LIN {X 0,Y 524.198,Z 429.088,A -85,B 0,C 180,E1 -4760.353,E2 -4760.353} C_VEL
LIN {X 0,Y 524.005,Z 439.005,A -85,B 0,C 180,E1 -4761.03,E2 -4761.03} C_VEL
LIN {X 0,Y 523.832,Z 446.958,A -85,B 0,C 180,E1 -4761.708,E2 -4761.708} C_VEL
LIN {X 0,Y 523.699,Z 454.397,A -85,B 0,C 180,E1 -4762.482,E2 -4762.482} C_VEL
LIN {X 0,Y 523.622,Z 461.025,A -85,B 0,C 180,E1 -4763.324,E2 -4763.324} C_VEL
LIN {X 0,Y 523.51,Z 467.877,A -85,B 0,C 180,E1 -4764.415,E2 -4764.415} C_VEL
LIN {X 0,Y 523.401,Z 472.538,A -85,B 0,C 180,E1 -4765.379,E2 -4765.379} C_VEL
LIN {X 0,Y 523.454,Z 475.573,A -85,B 0,C 180,E1 -4766.151,E2 -4766.151} C_VEL
LIN {X 0,Y 523.38,Z 477.92,A -85,B 0,C 180,E1 -4766.921,E2 -4766.921} C_VEL
LIN {X 0,Y 523.336,Z 479.685,A -85,B 0,C 180,E1 -4767.691,E2 -4767.691} C_VEL
LIN {X 0,Y 523.273,Z 480.952,A -85,B 0,C 180,E1 -4768.461,E2 -4768.461} C_VEL
LIN {X 0,Y 523.261,Z 481.745,A -85,B 0,C 180,E1 -4769.231,E2 -4769.231} C_VEL
LIN {X 0,Y 523.264,Z 482.047,A -85,B 0,C 180,E1 -4770,E2 -4770} C_VEL
LIN {X 0,Y 523.26,Z 481.751,A -85,B 0,C 180,E1 -4770.77,E2 -4770.77} C_VEL
LIN {X 0,Y 523.273,Z 480.966,A -85,B 0,C 180,E1 -4771.539,E2 -4771.539} C_VEL
LIN {X 0,Y 523.336,Z 479.706,A -85,B 0,C 180,E1 -4772.309,E2 -4772.309} C_VEL
LIN {X 0,Y 523.407,Z 476.783,A -85,B 0,C 180,E1 -4773.464,E2 -4773.464} C_VEL
LIN {X 0,Y 523.451,Z 474.115,A -85,B 0,C 180,E1 -4774.235,E2 -4774.235} C_VEL
LIN {X 0,Y 523.483,Z 468.893,A -85,B 0,C 180,E1 -4775.393,E2 -4775.393} C_VEL
LIN {X 0,Y 523.573,Z 462.971,A -85,B 0,C 180,E1 -4776.408,E2 -4776.408} C_VEL
LIN {X 0,Y 523.699,Z 456.194,A -85,B 0,C 180,E1 -4777.325,E2 -4777.325} C_VEL
LIN {X 0,Y 523.837,Z 448.092,A -85,B 0,C 180,E1 -4778.195,E2 -4778.195} C_VEL
LIN {X 0,Y 524.001,Z 440.358,A -85,B 0,C 180,E1 -4778.873,E2 -4778.873} C_VEL
LIN {X 0,Y 524.123,Z 432.228,A -85,B 0,C 180,E1 -4779.454,E2 -4779.454} C_VEL
LIN {X 0,Y 524.305,Z 423.801,A -85,B 0,C 180,E1 -4779.938,E2 -4779.938} C_VEL
LIN {X 0,Y 524.43,Z 415.18,A -85,B 0,C 180,E1 -4780.326,E2 -4780.326} C_VEL
LIN {X 0,Y 524.599,Z 404.889,A -85,B 0,C 180,E1 -4780.664,E2 -4780.664} C_VEL
LIN {X 0,Y 524.733,Z 390.891,A -85,B 0,C 180,E1 -4780.929,E2 -4780.929} C_VEL
LIN {X 0,Y 524.752,Z 329.083,A -85,B 0,C 180,E1 -4781.779,E2 -4781.779} C_VEL
LIN {X 0,Y 523.843,Z 320.89,A -85,B 0,C 180,E1 -4781.93,E2 -4781.93} C_VEL
LIN {X 0,Y 524.085,Z 303.68,A -85,B 0,C 180,E1 -4784.761,E2 -4784.761} C_VEL
LIN {X 0,Y 524.361,Z 286.918,A -85,B 0,C 180,E1 -4787.532,E2 -4787.532} C_VEL
LIN {X 0,Y 524.693,Z 269.864,A -85,B 0,C 180,E1 -4790.38,E2 -4790.38} C_VEL
LIN {X 0,Y 525.038,Z 257.174,A -85,B 0,C 180,E1 -4792.54,E2 -4792.54} C_VEL
LIN {X 0,Y 523.945,Z 250.036,A -85,B 0,C 180,E1 -4793.834,E2 -4793.834} C_VEL
LIN {X 0,Y 523.94,Z 250.03,A -85,B 0,C 180,E1 -4796.273,E2 -4796.273} C_VEL
LIN {X 0,Y 523.928,Z 250.031,A -85,B 0,C 180,E1 -4798.875,E2 -4798.875} C_VEL
LIN {X 0,Y 523.92,Z 250.04,A -85,B 0,C 180,E1 -4801.544,E2 -4801.544} C_VEL
LIN {X 0,Y 523.935,Z 250.029,A -85,B 0,C 180,E1 -4804.289,E2 -4804.289} C_VEL
LIN {X 0,Y 523.907,Z 250.035,A -85,B 0,C 180,E1 -4807.132,E2 -4807.132} C_VEL
LIN {X 0,Y 523.936,Z 250.03,A -85,B 0,C 180,E1 -4810.129,E2 -4810.129} C_VEL
LIN {X 0,Y 523.935,Z 250.028,A -85,B 0,C 180,E1 -4812.458,E2 -4812.458} C_VEL
LIN {X 0,Y 523.952,Z 250.032,A -85,B 0,C 180,E1 -4815.308,E2 -4815.308} C_VEL
LIN {X 0,Y 523.959,Z 250.026,A -85,B 0,C 180,E1 -4818.688,E2 -4818.688} C_VEL
LIN {X 0,Y 523.913,Z 250.035,A -85,B 0,C 180,E1 -4821.898,E2 -4821.898} C_VEL
LIN {X 0,Y 523.931,Z 250.03,A -85,B 0,C 180,E1 -4824.909,E2 -4824.909} C_VEL
LIN {X 0,Y 523.931,Z 250.036,A -85,B 0,C 180,E1 -4827.679,E2 -4827.679} C_VEL
LIN {X 0,Y 523.95,Z 250.027,A -85,B 0,C 180,E1 -4830.676,E2 -4830.676} C_VEL
LIN {X 0,Y 523.974,Z 250.03,A -85,B 0,C 180,E1 -4833.728,E2 -4833.728} C_VEL
LIN {X 0,Y 523.932,Z 250.03,A -85,B 0,C 180,E1 -4836.27,E2 -4836.27} C_VEL
LIN {X 0,Y 523.941,Z 250.028,A -85,B 0,C 180,E1 -4838.766,E2 -4838.766} C_VEL
LIN {X 0,Y 523.947,Z 250.032,A -85,B 0,C 180,E1 -4841.22,E2 -4841.22} C_VEL
LIN {X 0,Y 523.932,Z 250.037,A -85,B 0,C 180,E1 -4843.638,E2 -4843.638} C_VEL
LIN {X 0,Y 523.934,Z 250.031,A -85,B 0,C 180,E1 -4846.027,E2 -4846.027} C_VEL
LIN {X 0,Y 524.006,Z 250.02,A -85,B 0,C 180,E1 -4848.393,E2 -4848.393} C_VEL
LIN {X 0,Y 524.001,Z 250.029,A -85,B 0,C 180,E1 -4851.515,E2 -4851.515} C_VEL
LIN {X 0,Y 524.077,Z 250.011,A -85,B 0,C 180,E1 -4854.613,E2 -4854.613} C_VEL
LIN {X 0,Y 524.105,Z 250.015,A -85,B 0,C 180,E1 -4857.694,E2 -4857.694} C_VEL
LIN {X 0,Y 524.118,Z 250.006,A -85,B 0,C 180,E1 -4860.768,E2 -4860.768} C_VEL
LIN {X 0,Y 524.068,Z 250.015,A -85,B 0,C 180,E1 -4863.074,E2 -4863.074} C_VEL
LIN {X 0,Y 524.038,Z 250.017,A -85,B 0,C 180,E1 -4866.158,E2 -4866.158} C_VEL
LIN {X 0,Y 523.993,Z 250.026,A -85,B 0,C 180,E1 -4869.261,E2 -4869.261} C_VEL
LIN {X 0,Y 524.017,Z 250.025,A -85,B 0,C 180,E1 -4871.751,E2 -4871.751} C_VEL
LIN {X 0,Y 523.984,Z 250.025,A -85,B 0,C 180,E1 -4875.052,E2 -4875.052} C_VEL
LIN {X 0,Y 523.956,Z 250.029,A -85,B 0,C 180,E1 -4877.968,E2 -4877.968} C_VEL
LIN {X 0,Y 523.964,Z 250.025,A -85,B 0,C 180,E1 -4880.409,E2 -4880.409} C_VEL
LIN {X 0,Y 523.908,Z 250.033,A -85,B 0,C 180,E1 -4882.893,E2 -4882.893} C_VEL
LIN {X 0,Y 523.946,Z 250.034,A -85,B 0,C 180,E1 -4885.418,E2 -4885.418} C_VEL
LIN {X 0,Y 523.962,Z 250.029,A -85,B 0,C 180,E1 -4887.998,E2 -4887.998} C_VEL
LIN {X 0,Y 523.937,Z 250.029,A -85,B 0,C 180,E1 -4890.855,E2 -4890.855} C_VEL
LIN {X 0,Y 523.954,Z 250.033,A -85,B 0,C 180,E1 -4893.735,E2 -4893.735} C_VEL
LIN {X 0,Y 523.913,Z 250.032,A -85,B 0,C 180,E1 -4896.404,E2 -4896.404} C_VEL
LIN {X 0,Y 523.95,Z 250.03,A -85,B 0,C 180,E1 -4899.081,E2 -4899.081} C_VEL
LIN {X 0,Y 523.947,Z 250.029,A -85,B 0,C 180,E1 -4902.118,E2 -4902.118} C_VEL
LIN {X 0,Y 523.946,Z 250.033,A -85,B 0,C 180,E1 -4905.308,E2 -4905.308} C_VEL
LIN {X 0,Y 523.913,Z 250.033,A -85,B 0,C 180,E1 -4906.922,E2 -4906.922} C_VEL
LIN {X 0,Y 523.251,Z 250.123,A -85,B 0,C 180,E1 -4907.563,E2 -4907.563} C_VEL
LIN {X 0,Y 520.42,Z 250.473,A -85,B 0,C 180,E1 -4908.605,E2 -4908.605} C_VEL
LIN {X 0,Y 518.022,Z 250.772,A -85,B 0,C 180,E1 -4909.444,E2 -4909.444} C_VEL
LIN {X 0,Y 516.982,Z 250.898,A -85,B 0,C 180,E1 -4910.092,E2 -4910.092} C_VEL
LIN {X 0,Y 516.892,Z 250.907,A -85,B 0,C 180,E1 -4910.311,E2 -4910.311} C_VEL
LIN {X 0,Y 516.875,Z 250.914,A -85,B 0,C 180,E1 -4913.342,E2 -4913.342} C_VEL
LIN {X 0,Y 516.901,Z 250.907,A -85,B 0,C 180,E1 -4916.121,E2 -4916.121} C_VEL
LIN {X 0,Y 516.883,Z 250.909,A -85,B 0,C 180,E1 -4918.935,E2 -4918.935} C_VEL
LIN {X 0,Y 516.91,Z 250.913,A -85,B 0,C 180,E1 -4921.585,E2 -4921.585} C_VEL
LIN {X 0,Y 516.922,Z 250.904,A -85,B 0,C 180,E1 -4924.211,E2 -4924.211} C_VEL
LIN {X 0,Y 516.883,Z 250.908,A -85,B 0,C 180,E1 -4926.777,E2 -4926.777} C_VEL
LIN {X 0,Y 516.931,Z 250.908,A -85,B 0,C 180,E1 -4929.731,E2 -4929.731} C_VEL
LIN {X 0,Y 516.92,Z 250.903,A -85,B 0,C 180,E1 -4932.596,E2 -4932.596} C_VEL
LIN {X 0,Y 516.933,Z 250.903,A -85,B 0,C 180,E1 -4935.03,E2 -4935.03} C_VEL
LIN {X 0,Y 516.956,Z 250.9,A -85,B 0,C 180,E1 -4938.234,E2 -4938.234} C_VEL
LIN {X 0,Y 516.96,Z 250.904,A -85,B 0,C 180,E1 -4941.4,E2 -4941.4} C_VEL
LIN {X 0,Y 516.992,Z 250.901,A -85,B 0,C 180,E1 -4943.757,E2 -4943.757} C_VEL
LIN {X 0,Y 517.004,Z 250.893,A -85,B 0,C 180,E1 -4946.883,E2 -4946.883} C_VEL
LIN {X 0,Y 517.071,Z 250.887,A -85,B 0,C 180,E1 -4950,E2 -4950} C_VEL
LIN {X 0,Y 517.004,Z 250.895,A -85,B 0,C 180,E1 -4953.117,E2 -4953.117} C_VEL
LIN {X 0,Y 516.987,Z 250.896,A -85,B 0,C 180,E1 -4956.243,E2 -4956.243} C_VEL
LIN {X 0,Y 516.938,Z 250.906,A -85,B 0,C 180,E1 -4959.389,E2 -4959.389} C_VEL
LIN {X 0,Y 516.974,Z 250.902,A -85,B 0,C 180,E1 -4961.824,E2 -4961.824} C_VEL
LIN {X 0,Y 516.933,Z 250.905,A -85,B 0,C 180,E1 -4965.146,E2 -4965.146} C_VEL
LIN {X 0,Y 516.91,Z 250.906,A -85,B 0,C 180,E1 -4968.222,E2 -4968.222} C_VEL
LIN {X 0,Y 516.901,Z 250.906,A -85,B 0,C 180,E1 -4970.701,E2 -4970.701} C_VEL
LIN {X 0,Y 516.875,Z 250.911,A -85,B 0,C 180,E1 -4974.073,E2 -4974.073} C_VEL
LIN {X 0,Y 516.895,Z 250.906,A -85,B 0,C 180,E1 -4976.659,E2 -4976.659} C_VEL
LIN {X 0,Y 516.898,Z 250.913,A -85,B 0,C 180,E1 -4979.523,E2 -4979.523} C_VEL
LIN {X 0,Y 516.852,Z 250.914,A -85,B 0,C 180,E1 -4982.538,E2 -4982.538} C_VEL
LIN {X 0,Y 516.793,Z 251.018,A -85,B 0,C 180,E1 -4983.273,E2 -4983.273} C_VEL
LIN {X 0,Y 516.67,Z 263.387,A -85,B 0,C 180,E1 -4986.215,E2 -4986.215} C_VEL
LIN {X 0,Y 516.669,Z 266.59,A -85,B 0,C 180,E1 -4986.975,E2 -4986.975} C_VEL
LIN {X 0,Y 518.076,Z 276.047,A -85,B 0,C 180,E1 -4987.162,E2 -4987.162} C_VEL
LIN {X 0,Y 517.732,Z 341.991,A -85,B 0,C 180,E1 -4988.104,E2 -4988.104} C_VEL
LIN {X 0,Y 517.575,Z 351.656,A -85,B 0,C 180,E1 -4988.346,E2 -4988.346} C_VEL
LIN {X 0,Y 517.495,Z 362.877,A -85,B 0,C 180,E1 -4988.77,E2 -4988.77} C_VEL
LIN {X 0,Y 517.301,Z 373.42,A -85,B 0,C 180,E1 -4989.343,E2 -4989.343} C_VEL
LIN {X 0,Y 517.17,Z 382.012,A -85,B 0,C 180,E1 -4989.947,E2 -4989.947} C_VEL
LIN {X 0,Y 516.98,Z 389.085,A -85,B 0,C 180,E1 -4990.552,E2 -4990.552} C_VEL
LIN {X 0,Y 516.809,Z 395.968,A -85,B 0,C 180,E1 -4991.264,E2 -4991.264} C_VEL
LIN {X 0,Y 516.699,Z 402.062,A -85,B 0,C 180,E1 -4992.023,E2 -4992.023} C_VEL
LIN {X 0,Y 516.575,Z 407.636,A -85,B 0,C 180,E1 -4992.862,E2 -4992.862} C_VEL
LIN {X 0,Y 516.492,Z 411.725,A -85,B 0,C 180,E1 -4993.599,E2 -4993.599} C_VEL
LIN {X 0,Y 516.431,Z 415.602,A -85,B 0,C 180,E1 -4994.446,E2 -4994.446} C_VEL
LIN {X 0,Y 516.378,Z 417.937,A -85,B 0,C 180,E1 -4995.049,E2 -4995.049} C_VEL
LIN {X 0,Y 516.315,Z 421.216,A -85,B 0,C 180,E1 -4996.171,E2 -4996.171} C_VEL
LIN {X 0,Y 516.248,Z 423.364,A -85,B 0,C 180,E1 -4997.317,E2 -4997.317} C_VEL
LIN {X 0,Y 516.238,Z 424.442,A -85,B 0,C 180,E1 -4998.482,E2 -4998.482} C_VEL
LIN {X 0,Y 516.185,Z 424.428,A -85,B 0,C 180,E1 -4999.679,E2 -4999.679} C_VEL
LIN {X 0,Y 516.246,Z 423.25,A -85,B 0,C 180,E1 -5000.892,E2 -5000.892} C_VEL
LIN {X 0,Y 516.37,Z 420.424,A -85,B 0,C 180,E1 -5002.233,E2 -5002.233} C_VEL
LIN {X 0,Y 516.429,Z 416.582,A -85,B 0,C 180,E1 -5003.408,E2 -5003.408} C_VEL
LIN {X 0,Y 516.52,Z 411.822,A -85,B 0,C 180,E1 -5004.489,E2 -5004.489} C_VEL
LIN {X 0,Y 516.668,Z 405.27,A -85,B 0,C 180,E1 -5005.634,E2 -5005.634} C_VEL
LIN {X 0,Y 516.803,Z 398.188,A -85,B 0,C 180,E1 -5006.582,E2 -5006.582} C_VEL
LIN {X 0,Y 516.966,Z 391.83,A -85,B 0,C 180,E1 -5007.284,E2 -5007.284} C_VEL
LIN {X 0,Y 517.118,Z 384.016,A -85,B 0,C 180,E1 -5007.993,E2 -5007.993} C_VEL
LIN {X 0,Y 517.316,Z 377.131,A -85,B 0,C 180,E1 -5008.51,E2 -5008.51} C_VEL
LIN {X 0,Y 517.404,Z 368.457,A -85,B 0,C 180,E1 -5009.04,E2 -5009.04} C_VEL
LIN {X 0,Y 517.519,Z 360.001,A -85,B 0,C 180,E1 -5009.443,E2 -5009.443} C_VEL
LIN {X 0,Y 517.659,Z 350.143,A -85,B 0,C 180,E1 -5009.791,E2 -5009.791} C_VEL
LIN {X 0,Y 517.741,Z 340.557,A -85,B 0,C 180,E1 -5010.014,E2 -5010.014} C_VEL
LIN {X 0,Y 517.993,Z 274.3,A -85,B 0,C 180,E1 -5010.958,E2 -5010.958} C_VEL
LIN {X 0,Y 516.689,Z 266.184,A -85,B 0,C 180,E1 -5011.128,E2 -5011.128} C_VEL
LIN {X 0,Y 516.642,Z 252.977,A -85,B 0,C 180,E1 -5013.869,E2 -5013.869} C_VEL
LIN {X 0,Y 516.665,Z 250.944,A -85,B 0,C 180,E1 -5014.306,E2 -5014.306} C_VEL
LIN {X 0,Y 516.865,Z 250.914,A -85,B 0,C 180,E1 -5015.927,E2 -5015.927} C_VEL
LIN {X 0,Y 516.901,Z 250.909,A -85,B 0,C 180,E1 -5019.299,E2 -5019.299} C_VEL
LIN {X 0,Y 516.92,Z 250.911,A -85,B 0,C 180,E1 -5022.597,E2 -5022.597} C_VEL
LIN {X 0,Y 516.93,Z 250.904,A -85,B 0,C 180,E1 -5025.031,E2 -5025.031} C_VEL
LIN {X 0,Y 516.954,Z 250.904,A -85,B 0,C 180,E1 -5028.234,E2 -5028.234} C_VEL
LIN {X 0,Y 516.962,Z 250.898,A -85,B 0,C 180,E1 -5031.4,E2 -5031.4} C_VEL
LIN {X 0,Y 517.034,Z 250.896,A -85,B 0,C 180,E1 -5034.541,E2 -5034.541} C_VEL
LIN {X 0,Y 517.075,Z 250.883,A -85,B 0,C 180,E1 -5037.664,E2 -5037.664} C_VEL
LIN {X 0,Y 517.086,Z 250.886,A -85,B 0,C 180,E1 -5040.779,E2 -5040.779} C_VEL
LIN {X 0,Y 517.008,Z 250.893,A -85,B 0,C 180,E1 -5043.118,E2 -5043.118} C_VEL
LIN {X 0,Y 517.001,Z 250.898,A -85,B 0,C 180,E1 -5046.244,E2 -5046.244} C_VEL
LIN {X 0,Y 516.947,Z 250.899,A -85,B 0,C 180,E1 -5049.39,E2 -5049.39} C_VEL
LIN {X 0,Y 516.943,Z 250.9,A -85,B 0,C 180,E1 -5051.808,E2 -5051.808} C_VEL
LIN {X 0,Y 516.938,Z 250.901,A -85,B 0,C 180,E1 -5055.148,E2 -5055.148} C_VEL
LIN {X 0,Y 516.918,Z 250.907,A -85,B 0,C 180,E1 -5058.223,E2 -5058.223} C_VEL
LIN {X 0,Y 516.905,Z 250.908,A -85,B 0,C 180,E1 -5060.702,E2 -5060.702} C_VEL
LIN {X 0,Y 516.904,Z 250.908,A -85,B 0,C 180,E1 -5064.073,E2 -5064.073} C_VEL
LIN {X 0,Y 516.922,Z 250.909,A -85,B 0,C 180,E1 -5066.658,E2 -5066.658} C_VEL
LIN {X 0,Y 516.918,Z 250.9,A -85,B 0,C 180,E1 -5069.527,E2 -5069.527} C_VEL
LIN {X 0,Y 516.891,Z 250.912,A -85,B 0,C 180,E1 -5072.545,E2 -5072.545} C_VEL
LIN {X 0,Y 516.877,Z 250.909,A -85,B 0,C 180,E1 -5075.333,E2 -5075.333} C_VEL
LIN {X 0,Y 516.876,Z 250.909,A -85,B 0,C 180,E1 -5077.944,E2 -5077.944} C_VEL
LIN {X 0,Y 516.899,Z 250.911,A -85,B 0,C 180,E1 -5080.741,E2 -5080.741} C_VEL
LIN {X 0,Y 516.877,Z 250.909,A -85,B 0,C 180,E1 -5083.904,E2 -5083.904} C_VEL
LIN {X 0,Y 516.878,Z 250.912,A -85,B 0,C 180,E1 -5086.108,E2 -5086.108} C_VEL
LIN {X 0,Y 516.912,Z 250.912,A -85,B 0,C 180,E1 -5088.399,E2 -5088.399} C_VEL
LIN {X 0,Y 516.877,Z 250.909,A -85,B 0,C 180,E1 -5091.285,E2 -5091.285} C_VEL
LIN {X 0,Y 516.885,Z 250.913,A -85,B 0,C 180,E1 -5094.222,E2 -5094.222} C_VEL
LIN {X 0,Y 516.894,Z 250.909,A -85,B 0,C 180,E1 -5097.054,E2 -5097.054} C_VEL
LIN {X 0,Y 516.89,Z 250.909,A -85,B 0,C 180,E1 -5099.797,E2 -5099.797} C_VEL
LIN {X 0,Y 516.92,Z 250.913,A -85,B 0,C 180,E1 -5102.468,E2 -5102.468} C_VEL
LIN {X 0,Y 516.872,Z 250.914,A -85,B 0,C 180,E1 -5105.071,E2 -5105.071} C_VEL
LIN {X 0,Y 516.952,Z 251.04,A -85,B 0,C 180,E1 -5106.489,E2 -5106.489} C_VEL
LIN {X 0,Y 517.739,Z 256.188,A -85,B 0,C 180,E1 -5107.378,E2 -5107.378} C_VEL
LIN {X 0,Y 517.46,Z 271.126,A -85,B 0,C 180,E1 -5109.851,E2 -5109.851} C_VEL
LIN {X 0,Y 517.197,Z 289.02,A -85,B 0,C 180,E1 -5112.81,E2 -5112.81} C_VEL
LIN {X 0,Y 516.915,Z 308.666,A -85,B 0,C 180,E1 -5116.035,E2 -5116.035} C_VEL
LIN {X 0,Y 516.782,Z 320.167,A -85,B 0,C 180,E1 -5117.912,E2 -5117.912} C_VEL
LIN {X 0,Y 517.961,Z 332.425,A -85,B 0,C 180,E1 -5118.12,E2 -5118.12} C_VEL
LIN {X 0,Y 517.703,Z 397.435,A -85,B 0,C 180,E1 -5119.044,E2 -5119.044} C_VEL
LIN {X 0,Y 517.545,Z 406.634,A -85,B 0,C 180,E1 -5119.264,E2 -5119.264} C_VEL
LIN {X 0,Y 517.4,Z 415.707,A -85,B 0,C 180,E1 -5119.582,E2 -5119.582} C_VEL
LIN {X 0,Y 517.252,Z 425.04,A -85,B 0,C 180,E1 -5120.024,E2 -5120.024} C_VEL
LIN {X 0,Y 517.056,Z 434.644,A -85,B 0,C 180,E1 -5120.613,E2 -5120.613} C_VEL
LIN {X 0,Y 516.841,Z 444.446,A -85,B 0,C 180,E1 -5121.398,E2 -5121.398} C_VEL
LIN {X 0,Y 516.673,Z 452.231,A -85,B 0,C 180,E1 -5122.183,E2 -5122.183} C_VEL
LIN {X 0,Y 516.6,Z 458.647,A -85,B 0,C 180,E1 -5122.967,E2 -5122.967} C_VEL
LIN {X 0,Y 516.49,Z 465.165,A -85,B 0,C 180,E1 -5123.947,E2 -5123.947} C_VEL
LIN {X 0,Y 516.345,Z 470.359,A -85,B 0,C 180,E1 -5124.925,E2 -5124.925} C_VEL
LIN {X 0,Y 516.382,Z 475.166,A -85,B 0,C 180,E1 -5126.098,E2 -5126.098} C_VEL
LIN {X 0,Y 516.294,Z 477.517,A -85,B 0,C 180,E1 -5126.879,E2 -5126.879} C_VEL
LIN {X 0,Y 516.263,Z 479.288,A -85,B 0,C 180,E1 -5127.66,E2 -5127.66} C_VEL
LIN {X 0,Y 516.191,Z 480.556,A -85,B 0,C 180,E1 -5128.44,E2 -5128.44} C_VEL
LIN {X 0,Y 516.171,Z 481.352,A -85,B 0,C 180,E1 -5129.22,E2 -5129.22} C_VEL
LIN {X 0,Y 516.175,Z 481.656,A -85,B 0,C 180,E1 -5130,E2 -5130} C_VEL
LIN {X 0,Y 516.17,Z 481.362,A -85,B 0,C 180,E1 -5130.78,E2 -5130.78} C_VEL
LIN {X 0,Y 516.191,Z 480.576,A -85,B 0,C 180,E1 -5131.561,E2 -5131.561} C_VEL
LIN {X 0,Y 516.263,Z 479.316,A -85,B 0,C 180,E1 -5132.341,E2 -5132.341} C_VEL
LIN {X 0,Y 516.325,Z 476.391,A -85,B 0,C 180,E1 -5133.512,E2 -5133.512} C_VEL
LIN {X 0,Y 516.359,Z 473.719,A -85,B 0,C 180,E1 -5134.293,E2 -5134.293} C_VEL
LIN {X 0,Y 516.42,Z 468.494,A -85,B 0,C 180,E1 -5135.467,E2 -5135.467} C_VEL
LIN {X 0,Y 516.475,Z 463.247,A -85,B 0,C 180,E1 -5136.384,E2 -5136.384} C_VEL
LIN {X 0,Y 516.622,Z 455.778,A -85,B 0,C 180,E1 -5137.425,E2 -5137.425} C_VEL
LIN {X 0,Y 516.753,Z 447.666,A -85,B 0,C 180,E1 -5138.309,E2 -5138.309} C_VEL
LIN {X 0,Y 516.941,Z 439.922,A -85,B 0,C 180,E1 -5138.995,E2 -5138.995} C_VEL
LIN {X 0,Y 517.091,Z 431.782,A -85,B 0,C 180,E1 -5139.584,E2 -5139.584} C_VEL
LIN {X 0,Y 517.287,Z 423.339,A -85,B 0,C 180,E1 -5140.074,E2 -5140.074} C_VEL
LIN {X 0,Y 517.434,Z 414.697,A -85,B 0,C 180,E1 -5140.467,E2 -5140.467} C_VEL
LIN {X 0,Y 517.611,Z 404.371,A -85,B 0,C 180,E1 -5140.809,E2 -5140.809} C_VEL
LIN {X 0,Y 517.77,Z 390.507,A -85,B 0,C 180,E1 -5141.074,E2 -5141.074} C_VEL
LIN {X 0,Y 517.859,Z 330.1,A -85,B 0,C 180,E1 -5141.919,E2 -5141.919} C_VEL
LIN {X 0,Y 516.793,Z 320.495,A -85,B 0,C 180,E1 -5142.099,E2 -5142.099} C_VEL
LIN {X 0,Y 517.047,Z 303.305,A -85,B 0,C 180,E1 -5144.967,E2 -5144.967} C_VEL
LIN {X 0,Y 517.344,Z 286.97,A -85,B 0,C 180,E1 -5147.711,E2 -5147.711} C_VEL
LIN {X 0,Y 517.838,Z 268.372,A -85,B 0,C 180,E1 -5150.87,E2 -5150.87} C_VEL
LIN {X 0,Y 517.946,Z 256.759,A -85,B 0,C 180,E1 -5152.882,E2 -5152.882} C_VEL
LIN {X 0,Y 516.9,Z 250.913,A -85,B 0,C 180,E1 -5153.966,E2 -5153.966} C_VEL
LIN {X 0,Y 516.907,Z 250.906,A -85,B 0,C 180,E1 -5156.658,E2 -5156.658} C_VEL
LIN {X 0,Y 516.91,Z 250.913,A -85,B 0,C 180,E1 -5159.523,E2 -5159.523} C_VEL
LIN {X 0,Y 516.895,Z 250.905,A -85,B 0,C 180,E1 -5162.543,E2 -5162.543} C_VEL
LIN {X 0,Y 516.87,Z 250.915,A -85,B 0,C 180,E1 -5165.33,E2 -5165.33} C_VEL
LIN {X 0,Y 516.878,Z 250.911,A -85,B 0,C 180,E1 -5167.942,E2 -5167.942} C_VEL
LIN {X 0,Y 516.883,Z 250.907,A -85,B 0,C 180,E1 -5170.741,E2 -5170.741} C_VEL
LIN {X 0,Y 516.882,Z 250.908,A -85,B 0,C 180,E1 -5172.831,E2 -5172.831} C_VEL
LIN {X 0,Y 516.921,Z 250.904,A -85,B 0,C 180,E1 -5175.009,E2 -5175.009} C_VEL
LIN {X 0,Y 516.915,Z 250.903,A -85,B 0,C 180,E1 -5178.398,E2 -5178.398} C_VEL
LIN {X 0,Y 516.878,Z 250.913,A -85,B 0,C 180,E1 -5181.284,E2 -5181.284} C_VEL
LIN {X 0,Y 516.885,Z 250.908,A -85,B 0,C 180,E1 -5184.22,E2 -5184.22} C_VEL
LIN {X 0,Y 516.891,Z 250.909,A -85,B 0,C 180,E1 -5187.052,E2 -5187.052} C_VEL
LIN {X 0,Y 516.888,Z 250.912,A -85,B 0,C 180,E1 -5189.796,E2 -5189.796} C_VEL
LIN {X 0,Y 516.926,Z 250.902,A -85,B 0,C 180,E1 -5192.467,E2 -5192.467} C_VEL
LIN {X 0,Y 516.908,Z 250.907,A -85,B 0,C 180,E1 -5195.071,E2 -5195.071} C_VEL
LIN {X 0,Y 516.881,Z 250.907,A -85,B 0,C 180,E1 -5198.462,E2 -5198.462} C_VEL
LIN {X 0,Y 516.898,Z 250.907,A -85,B 0,C 180,E1 -5200.954,E2 -5200.954} C_VEL
LIN {X 0,Y 516.909,Z 250.911,A -85,B 0,C 180,E1 -5203.41,E2 -5203.41} C_VEL
LIN {X 0,Y 516.889,Z 250.911,A -85,B 0,C 180,E1 -5205.833,E2 -5205.833} C_VEL
LIN {X 0,Y 516.96,Z 250.898,A -85,B 0,C 180,E1 -5208.233,E2 -5208.233} C_VEL
LIN {X 0,Y 516.965,Z 250.904,A -85,B 0,C 180,E1 -5211.399,E2 -5211.399} C_VEL
LIN {X 0,Y 517.004,Z 250.898,A -85,B 0,C 180,E1 -5213.756,E2 -5213.756} C_VEL
LIN {X 0,Y 517.077,Z 250.891,A -85,B 0,C 180,E1 -5217.662,E2 -5217.662} C_VEL
LIN {X 0,Y 517.088,Z 250.882,A -85,B 0,C 180,E1 -5220.778,E2 -5220.778} C_VEL
LIN {X 0,Y 517.009,Z 250.895,A -85,B 0,C 180,E1 -5223.116,E2 -5223.116} C_VEL
LIN {X 0,Y 517.002,Z 250.893,A -85,B 0,C 180,E1 -5226.243,E2 -5226.243} C_VEL
LIN {X 0,Y 516.947,Z 250.906,A -85,B 0,C 180,E1 -5229.389,E2 -5229.389} C_VEL
LIN {X 0,Y 516.976,Z 250.901,A -85,B 0,C 180,E1 -5231.823,E2 -5231.823} C_VEL
LIN {X 0,Y 516.936,Z 250.904,A -85,B 0,C 180,E1 -5235.146,E2 -5235.146} C_VEL
LIN {X 0,Y 516.918,Z 250.904,A -85,B 0,C 180,E1 -5238.222,E2 -5238.222} C_VEL
LIN {X 0,Y 516.904,Z 250.905,A -85,B 0,C 180,E1 -5240.701,E2 -5240.701} C_VEL
LIN {X 0,Y 516.902,Z 250.907,A -85,B 0,C 180,E1 -5244.071,E2 -5244.071} C_VEL
LIN {X 0,Y 516.92,Z 250.903,A -85,B 0,C 180,E1 -5246.657,E2 -5246.657} C_VEL
LIN {X 0,Y 516.902,Z 250.913,A -85,B 0,C 180,E1 -5249.523,E2 -5249.523} C_VEL
LIN {X 0,Y 516.892,Z 250.906,A -85,B 0,C 180,E1 -5252.544,E2 -5252.544} C_VEL
LIN {X 0,Y 516.875,Z 250.914,A -85,B 0,C 180,E1 -5255.332,E2 -5255.332} C_VEL
LIN {X 0,Y 516.872,Z 250.912,A -85,B 0,C 180,E1 -5257.943,E2 -5257.943} C_VEL
LIN {X 0,Y 516.885,Z 250.907,A -85,B 0,C 180,E1 -5260.74,E2 -5260.74} C_VEL
LIN {X 0,Y 516.872,Z 250.913,A -85,B 0,C 180,E1 -5263.893,E2 -5263.893} C_VEL
LIN {X 0,Y 516.873,Z 250.911,A -85,B 0,C 180,E1 -5266.107,E2 -5266.107} C_VEL
LIN {X 0,Y 516.894,Z 250.911,A -85,B 0,C 180,E1 -5269.26,E2 -5269.26} C_VEL
LIN {X 0,Y 516.892,Z 250.907,A -85,B 0,C 180,E1 -5270.311,E2 -5270.311} C_VEL
LIN {X 0,Y 516.211,Z 250.993,A -85,B 0,C 180,E1 -5270.962,E2 -5270.962} C_VEL
LIN {X 0,Y 513.358,Z 251.356,A -85,B 0,C 180,E1 -5272.017,E2 -5272.017} C_VEL
LIN {X 0,Y 510.949,Z 251.66,A -85,B 0,C 180,E1 -5272.867,E2 -5272.867} C_VEL
LIN {X 0,Y 509.909,Z 251.786,A -85,B 0,C 180,E1 -5273.524,E2 -5273.524} C_VEL
LIN {X 0,Y 509.82,Z 251.794,A -85,B 0,C 180,E1 -5273.746,E2 -5273.746} C_VEL
LIN {X 0,Y 509.852,Z 251.783,A -85,B 0,C 180,E1 -5276.539,E2 -5276.539} C_VEL
LIN {X 0,Y 509.837,Z 251.79,A -85,B 0,C 180,E1 -5279.334,E2 -5279.334} C_VEL
LIN {X 0,Y 509.885,Z 251.782,A -85,B 0,C 180,E1 -5282.054,E2 -5282.054} C_VEL
LIN {X 0,Y 509.869,Z 251.781,A -85,B 0,C 180,E1 -5284.704,E2 -5284.704} C_VEL
LIN {X 0,Y 509.857,Z 251.789,A -85,B 0,C 180,E1 -5287.447,E2 -5287.447} C_VEL
LIN {X 0,Y 509.908,Z 251.782,A -85,B 0,C 180,E1 -5289.845,E2 -5289.845} C_VEL
LIN {X 0,Y 509.876,Z 251.784,A -85,B 0,C 180,E1 -5293.175,E2 -5293.175} C_VEL
LIN {X 0,Y 509.855,Z 251.792,A -85,B 0,C 180,E1 -5295.634,E2 -5295.634} C_VEL
LIN {X 0,Y 509.908,Z 251.777,A -85,B 0,C 180,E1 -5298.874,E2 -5298.874} C_VEL
LIN {X 0,Y 509.942,Z 251.775,A -85,B 0,C 180,E1 -5302.078,E2 -5302.078} C_VEL
LIN {X 0,Y 509.969,Z 251.769,A -85,B 0,C 180,E1 -5304.464,E2 -5304.464} C_VEL
LIN {X 0,Y 510.043,Z 251.768,A -85,B 0,C 180,E1 -5307.631,E2 -5307.631} C_VEL
LIN {X 0,Y 510.042,Z 251.763,A -85,B 0,C 180,E1 -5310,E2 -5310} C_VEL
LIN {X 0,Y 510.042,Z 251.76,A -85,B 0,C 180,E1 -5312.369,E2 -5312.369} C_VEL
LIN {X 0,Y 509.964,Z 251.777,A -85,B 0,C 180,E1 -5315.536,E2 -5315.536} C_VEL
LIN {X 0,Y 509.94,Z 251.777,A -85,B 0,C 180,E1 -5317.921,E2 -5317.921} C_VEL
LIN {X 0,Y 509.911,Z 251.779,A -85,B 0,C 180,E1 -5321.125,E2 -5321.125} C_VEL
LIN {X 0,Y 509.85,Z 251.784,A -85,B 0,C 180,E1 -5324.366,E2 -5324.366} C_VEL
LIN {X 0,Y 509.881,Z 251.788,A -85,B 0,C 180,E1 -5327.652,E2 -5327.652} C_VEL
LIN {X 0,Y 509.875,Z 251.781,A -85,B 0,C 180,E1 -5330.401,E2 -5330.401} C_VEL
LIN {X 0,Y 509.808,Z 251.796,A -85,B 0,C 180,E1 -5333.564,E2 -5333.564} C_VEL
LIN {X 0,Y 509.874,Z 251.781,A -85,B 0,C 180,E1 -5336.372,E2 -5336.372} C_VEL
LIN {X 0,Y 509.859,Z 251.783,A -85,B 0,C 180,E1 -5338.844,E2 -5338.844} C_VEL
LIN {X 0,Y 509.798,Z 251.799,A -85,B 0,C 180,E1 -5341.591,E2 -5341.591} C_VEL
LIN {X 0,Y 509.776,Z 251.866,A -85,B 0,C 180,E1 -5343.225,E2 -5343.225} C_VEL
LIN {X 0,Y 509.658,Z 265.006,A -85,B 0,C 180,E1 -5346.366,E2 -5346.366} C_VEL
LIN {X 0,Y 509.675,Z 266.94,A -85,B 0,C 180,E1 -5346.822,E2 -5346.822} C_VEL
LIN {X 0,Y 511.144,Z 277.27,A -85,B 0,C 180,E1 -5347.013,E2 -5347.013} C_VEL
LIN {X 0,Y 510.77,Z 342.356,A -85,B 0,C 180,E1 -5347.958,E2 -5347.958} C_VEL
LIN {X 0,Y 510.604,Z 352.172,A -85,B 0,C 180,E1 -5348.207,E2 -5348.207} C_VEL
LIN {X 0,Y 510.517,Z 362.634,A -85,B 0,C 180,E1 -5348.606,E2 -5348.606} C_VEL
LIN {X 0,Y 510.336,Z 373.075,A -85,B 0,C 180,E1 -5349.166,E2 -5349.166} C_VEL
LIN {X 0,Y 510.187,Z 381.972,A -85,B 0,C 180,E1 -5349.792,E2 -5349.792} C_VEL
LIN {X 0,Y 509.997,Z 388.709,A -85,B 0,C 180,E1 -5350.366,E2 -5350.366} C_VEL
LIN {X 0,Y 509.803,Z 395.325,A -85,B 0,C 180,E1 -5351.04,E2 -5351.04} C_VEL
LIN {X 0,Y 509.677,Z 402.06,A -85,B 0,C 180,E1 -5351.876,E2 -5351.876} C_VEL
LIN {X 0,Y 509.521,Z 407.974,A -85,B 0,C 180,E1 -5352.772,E2 -5352.772} C_VEL
LIN {X 0,Y 509.441,Z 412.513,A -85,B 0,C 180,E1 -5353.611,E2 -5353.611} C_VEL
LIN {X 0,Y 509.361,Z 416.318,A -85,B 0,C 180,E1 -5354.472,E2 -5354.472} C_VEL
LIN {X 0,Y 509.286,Z 419.183,A -85,B 0,C 180,E1 -5355.27,E2 -5355.27} C_VEL
LIN {X 0,Y 509.22,Z 422.075,A -85,B 0,C 180,E1 -5356.366,E2 -5356.366} C_VEL
LIN {X 0,Y 509.151,Z 423.932,A -85,B 0,C 180,E1 -5357.441,E2 -5357.441} C_VEL
LIN {X 0,Y 509.148,Z 424.847,A -85,B 0,C 180,E1 -5358.506,E2 -5358.506} C_VEL
LIN {X 0,Y 509.114,Z 424.873,A -85,B 0,C 180,E1 -5359.55,E2 -5359.55} C_VEL
LIN {X 0,Y 509.151,Z 423.998,A -85,B 0,C 180,E1 -5360.621,E2 -5360.621} C_VEL
LIN {X 0,Y 509.229,Z 421.828,A -85,B 0,C 180,E1 -5361.874,E2 -5361.874} C_VEL
LIN {X 0,Y 509.347,Z 418.159,A -85,B 0,C 180,E1 -5363.156,E2 -5363.156} C_VEL
LIN {X 0,Y 509.432,Z 414.53,A -85,B 0,C 180,E1 -5364.078,E2 -5364.078} C_VEL
LIN {X 0,Y 509.503,Z 409.488,A -85,B 0,C 180,E1 -5365.08,E2 -5365.08} C_VEL
LIN {X 0,Y 509.65,Z 403.272,A -85,B 0,C 180,E1 -5366.062,E2 -5366.062} C_VEL
LIN {X 0,Y 509.768,Z 398.115,A -85,B 0,C 180,E1 -5366.738,E2 -5366.738} C_VEL
LIN {X 0,Y 509.966,Z 391.25,A -85,B 0,C 180,E1 -5367.49,E2 -5367.49} C_VEL
LIN {X 0,Y 510.151,Z 383.313,A -85,B 0,C 180,E1 -5368.202,E2 -5368.202} C_VEL
LIN {X 0,Y 510.338,Z 374.951,A -85,B 0,C 180,E1 -5368.809,E2 -5368.809} C_VEL
LIN {X 0,Y 510.492,Z 365.009,A -85,B 0,C 180,E1 -5369.378,E2 -5369.378} C_VEL
LIN {X 0,Y 510.665,Z 353.488,A -85,B 0,C 180,E1 -5369.846,E2 -5369.846} C_VEL
LIN {X 0,Y 510.745,Z 343.219,A -85,B 0,C 180,E1 -5370.118,E2 -5370.118} C_VEL
LIN {X 0,Y 511.073,Z 274.922,A -85,B 0,C 180,E1 -5371.118,E2 -5371.118} C_VEL
LIN {X 0,Y 509.646,Z 266.492,A -85,B 0,C 180,E1 -5371.295,E2 -5371.295} C_VEL
LIN {X 0,Y 509.611,Z 253.23,A -85,B 0,C 180,E1 -5374.034,E2 -5374.034} C_VEL
LIN {X 0,Y 509.638,Z 251.819,A -85,B 0,C 180,E1 -5374.364,E2 -5374.364} C_VEL
LIN {X 0,Y 509.806,Z 251.798,A -85,B 0,C 180,E1 -5376.436,E2 -5376.436} C_VEL
LIN {X 0,Y 509.905,Z 251.781,A -85,B 0,C 180,E1 -5379.845,E2 -5379.845} C_VEL
LIN {X 0,Y 509.876,Z 251.783,A -85,B 0,C 180,E1 -5383.175,E2 -5383.175} C_VEL
LIN {X 0,Y 509.853,Z 251.784,A -85,B 0,C 180,E1 -5385.635,E2 -5385.635} C_VEL
LIN {X 0,Y 509.907,Z 251.781,A -85,B 0,C 180,E1 -5388.875,E2 -5388.875} C_VEL
LIN {X 0,Y 509.942,Z 251.776,A -85,B 0,C 180,E1 -5392.079,E2 -5392.079} C_VEL
LIN {X 0,Y 509.984,Z 251.775,A -85,B 0,C 180,E1 -5394.465,E2 -5394.465} C_VEL
LIN {X 0,Y 510.046,Z 251.758,A -85,B 0,C 180,E1 -5397.632,E2 -5397.632} C_VEL
LIN {X 0,Y 510.056,Z 251.762,A -85,B 0,C 180,E1 -5400.79,E2 -5400.79} C_VEL
LIN {X 0,Y 509.95,Z 251.772,A -85,B 0,C 180,E1 -5403.161,E2 -5403.161} C_VEL
LIN {X 0,Y 509.97,Z 251.775,A -85,B 0,C 180,E1 -5406.33,E2 -5406.33} C_VEL
LIN {X 0,Y 509.909,Z 251.781,A -85,B 0,C 180,E1 -5408.721,E2 -5408.721} C_VEL
LIN {X 0,Y 509.895,Z 251.779,A -85,B 0,C 180,E1 -5411.932,E2 -5411.932} C_VEL
LIN {X 0,Y 509.885,Z 251.779,A -85,B 0,C 180,E1 -5415.243,E2 -5415.243} C_VEL
LIN {X 0,Y 509.881,Z 251.78,A -85,B 0,C 180,E1 -5418.002,E2 -5418.002} C_VEL
LIN {X 0,Y 509.843,Z 251.784,A -85,B 0,C 180,E1 -5421.002,E2 -5421.002} C_VEL
LIN {X 0,Y 509.829,Z 251.786,A -85,B 0,C 180,E1 -5423.564,E2 -5423.564} C_VEL
LIN {X 0,Y 509.907,Z 251.781,A -85,B 0,C 180,E1 -5426.38,E2 -5426.38} C_VEL
LIN {X 0,Y 509.879,Z 251.781,A -85,B 0,C 180,E1 -5428.845,E2 -5428.845} C_VEL
LIN {X 0,Y 509.816,Z 251.788,A -85,B 0,C 180,E1 -5431.591,E2 -5431.591} C_VEL
LIN {X 0,Y 509.848,Z 251.789,A -85,B 0,C 180,E1 -5434.414,E2 -5434.414} C_VEL
LIN {X 0,Y 509.814,Z 251.786,A -85,B 0,C 180,E1 -5437.341,E2 -5437.341} C_VEL
LIN {X 0,Y 509.856,Z 251.79,A -85,B 0,C 180,E1 -5440.381,E2 -5440.381} C_VEL
LIN {X 0,Y 509.818,Z 251.788,A -85,B 0,C 180,E1 -5443.063,E2 -5443.063} C_VEL
LIN {X 0,Y 509.826,Z 251.788,A -85,B 0,C 180,E1 -5445.793,E2 -5445.793} C_VEL
LIN {X 0,Y 509.853,Z 251.79,A -85,B 0,C 180,E1 -5448.576,E2 -5448.576} C_VEL
LIN {X 0,Y 509.847,Z 251.785,A -85,B 0,C 180,E1 -5451.787,E2 -5451.787} C_VEL
LIN {X 0,Y 509.84,Z 251.792,A -85,B 0,C 180,E1 -5454.624,E2 -5454.624} C_VEL
LIN {X 0,Y 509.861,Z 251.783,A -85,B 0,C 180,E1 -5457.482,E2 -5457.482} C_VEL
LIN {X 0,Y 509.857,Z 251.791,A -85,B 0,C 180,E1 -5460.275,E2 -5460.275} C_VEL
LIN {X 0,Y 509.879,Z 251.785,A -85,B 0,C 180,E1 -5462.945,E2 -5462.945} C_VEL
LIN {X 0,Y 509.875,Z 251.79,A -85,B 0,C 180,E1 -5466.332,E2 -5466.332} C_VEL
LIN {X 0,Y 510.731,Z 257.328,A -85,B 0,C 180,E1 -5467.338,E2 -5467.338} C_VEL
LIN {X 0,Y 510.43,Z 272.398,A -85,B 0,C 180,E1 -5469.866,E2 -5469.866} C_VEL
LIN {X 0,Y 510.166,Z 289.778,A -85,B 0,C 180,E1 -5472.772,E2 -5472.772} C_VEL
LIN {X 0,Y 509.859,Z 309.46,A -85,B 0,C 180,E1 -5476.042,E2 -5476.042} C_VEL
LIN {X 0,Y 509.697,Z 319.753,A -85,B 0,C 180,E1 -5477.744,E2 -5477.744} C_VEL
LIN {X 0,Y 511.021,Z 333.154,A -85,B 0,C 180,E1 -5477.973,E2 -5477.973} C_VEL
LIN {X 0,Y 510.735,Z 398.066,A -85,B 0,C 180,E1 -5478.918,E2 -5478.918} C_VEL
LIN {X 0,Y 510.513,Z 408.55,A -85,B 0,C 180,E1 -5479.189,E2 -5479.189} C_VEL
LIN {X 0,Y 510.265,Z 420.767,A -85,B 0,C 180,E1 -5479.686,E2 -5479.686} C_VEL
LIN {X 0,Y 510.129,Z 429.626,A -85,B 0,C 180,E1 -5480.184,E2 -5480.184} C_VEL
LIN {X 0,Y 509.971,Z 438.069,A -85,B 0,C 180,E1 -5480.782,E2 -5480.782} C_VEL
LIN {X 0,Y 509.729,Z 446.048,A -85,B 0,C 180,E1 -5481.477,E2 -5481.477} C_VEL
LIN {X 0,Y 509.571,Z 453.51,A -85,B 0,C 180,E1 -5482.272,E2 -5482.272} C_VEL
LIN {X 0,Y 509.465,Z 461.52,A -85,B 0,C 180,E1 -5483.33,E2 -5483.33} C_VEL
LIN {X 0,Y 509.335,Z 468.005,A -85,B 0,C 180,E1 -5484.458,E2 -5484.458} C_VEL
LIN {X 0,Y 509.25,Z 473.254,A -85,B 0,C 180,E1 -5485.647,E2 -5485.647} C_VEL
LIN {X 0,Y 509.247,Z 475.941,A -85,B 0,C 180,E1 -5486.44,E2 -5486.44} C_VEL
LIN {X 0,Y 509.192,Z 478.891,A -85,B 0,C 180,E1 -5487.627,E2 -5487.627} C_VEL
LIN {X 0,Y 509.111,Z 480.161,A -85,B 0,C 180,E1 -5488.418,E2 -5488.418} C_VEL
LIN {X 0,Y 509.083,Z 480.958,A -85,B 0,C 180,E1 -5489.209,E2 -5489.209} C_VEL
LIN {X 0,Y 509.086,Z 481.265,A -85,B 0,C 180,E1 -5490,E2 -5490} C_VEL
LIN {X 0,Y 509.083,Z 480.972,A -85,B 0,C 180,E1 -5490.791,E2 -5490.791} C_VEL
LIN {X 0,Y 509.111,Z 480.187,A -85,B 0,C 180,E1 -5491.582,E2 -5491.582} C_VEL
LIN {X 0,Y 509.192,Z 478.926,A -85,B 0,C 180,E1 -5492.373,E2 -5492.373} C_VEL
LIN {X 0,Y 509.247,Z 475.999,A -85,B 0,C 180,E1 -5493.561,E2 -5493.561} C_VEL
LIN {X 0,Y 509.25,Z 473.323,A -85,B 0,C 180,E1 -5494.353,E2 -5494.353} C_VEL
LIN {X 0,Y 509.335,Z 468.094,A -85,B 0,C 180,E1 -5495.543,E2 -5495.543} C_VEL
LIN {X 0,Y 509.452,Z 461.709,A -85,B 0,C 180,E1 -5496.657,E2 -5496.657} C_VEL
LIN {X 0,Y 509.572,Z 453.649,A -85,B 0,C 180,E1 -5497.728,E2 -5497.728} C_VEL
LIN {X 0,Y 509.771,Z 446.216,A -85,B 0,C 180,E1 -5498.523,E2 -5498.523} C_VEL
LIN {X 0,Y 509.974,Z 438.254,A -85,B 0,C 180,E1 -5499.219,E2 -5499.219} C_VEL
LIN {X 0,Y 510.177,Z 428.323,A -85,B 0,C 180,E1 -5499.915,E2 -5499.915} C_VEL
LIN {X 0,Y 510.405,Z 417.85,A -85,B 0,C 180,E1 -5500.462,E2 -5500.462} C_VEL
LIN {X 0,Y 510.564,Z 407.168,A -85,B 0,C 180,E1 -5500.86,E2 -5500.86} C_VEL
LIN {X 0,Y 510.729,Z 398.387,A -85,B 0,C 180,E1 -5501.082,E2 -5501.082} C_VEL
LIN {X 0,Y 510.873,Z 330.339,A -85,B 0,C 180,E1 -5502.075,E2 -5502.075} C_VEL
LIN {X 0,Y 509.713,Z 320.122,A -85,B 0,C 180,E1 -5502.27,E2 -5502.27} C_VEL
LIN {X 0,Y 509.983,Z 304.129,A -85,B 0,C 180,E1 -5504.974,E2 -5504.974} C_VEL
LIN {X 0,Y 510.338,Z 286.985,A -85,B 0,C 180,E1 -5507.896,E2 -5507.896} C_VEL
LIN {X 0,Y 510.862,Z 269.255,A -85,B 0,C 180,E1 -5510.958,E2 -5510.958} C_VEL
LIN {X 0,Y 511.025,Z 258.39,A -85,B 0,C 180,E1 -5512.863,E2 -5512.863} C_VEL
LIN {X 0,Y 509.853,Z 251.789,A -85,B 0,C 180,E1 -5514.102,E2 -5514.102} C_VEL
LIN {X 0,Y 509.874,Z 251.785,A -85,B 0,C 180,E1 -5517.056,E2 -5517.056} C_VEL
LIN {X 0,Y 509.857,Z 251.788,A -85,B 0,C 180,E1 -5519.751,E2 -5519.751} C_VEL
LIN {X 0,Y 509.873,Z 251.781,A -85,B 0,C 180,E1 -5522.774,E2 -5522.774} C_VEL
LIN {X 0,Y 509.829,Z 251.794,A -85,B 0,C 180,E1 -5525.579,E2 -5525.579} C_VEL
LIN {X 0,Y 509.848,Z 251.784,A -85,B 0,C 180,E1 -5528.338,E2 -5528.338} C_VEL
LIN {X 0,Y 509.855,Z 251.79,A -85,B 0,C 180,E1 -5531.425,E2 -5531.425} C_VEL
LIN {X 0,Y 509.855,Z 251.783,A -85,B 0,C 180,E1 -5534.667,E2 -5534.667} C_VEL
LIN {X 0,Y 509.856,Z 251.784,A -85,B 0,C 180,E1 -5538.102,E2 -5538.102} C_VEL
LIN {X 0,Y 509.844,Z 251.784,A -85,B 0,C 180,E1 -5540.647,E2 -5540.647} C_VEL
LIN {X 0,Y 509.832,Z 251.793,A -85,B 0,C 180,E1 -5543.647,E2 -5543.647} C_VEL
LIN {X 0,Y 509.857,Z 251.782,A -85,B 0,C 180,E1 -5546.539,E2 -5546.539} C_VEL
LIN {X 0,Y 509.841,Z 251.79,A -85,B 0,C 180,E1 -5549.334,E2 -5549.334} C_VEL
LIN {X 0,Y 509.891,Z 251.78,A -85,B 0,C 180,E1 -5552.054,E2 -5552.054} C_VEL
LIN {X 0,Y 509.874,Z 251.78,A -85,B 0,C 180,E1 -5554.703,E2 -5554.703} C_VEL
LIN {X 0,Y 509.832,Z 251.793,A -85,B 0,C 180,E1 -5557.454,E2 -5557.454} C_VEL
LIN {X 0,Y 509.912,Z 251.78,A -85,B 0,C 180,E1 -5559.844,E2 -5559.844} C_VEL
LIN {X 0,Y 509.879,Z 251.783,A -85,B 0,C 180,E1 -5563.174,E2 -5563.174} C_VEL
LIN {X 0,Y 509.858,Z 251.79,A -85,B 0,C 180,E1 -5565.633,E2 -5565.633} C_VEL
LIN {X 0,Y 509.907,Z 251.777,A -85,B 0,C 180,E1 -5568.874,E2 -5568.874} C_VEL
LIN {X 0,Y 509.946,Z 251.773,A -85,B 0,C 180,E1 -5572.078,E2 -5572.078} C_VEL
LIN {X 0,Y 509.976,Z 251.768,A -85,B 0,C 180,E1 -5574.464,E2 -5574.464} C_VEL
LIN {X 0,Y 510.048,Z 251.767,A -85,B 0,C 180,E1 -5577.63,E2 -5577.63} C_VEL
LIN {X 0,Y 510.058,Z 251.758,A -85,B 0,C 180,E1 -5580.789,E2 -5580.789} C_VEL
LIN {X 0,Y 509.951,Z 251.774,A -85,B 0,C 180,E1 -5583.159,E2 -5583.159} C_VEL
LIN {X 0,Y 509.971,Z 251.769,A -85,B 0,C 180,E1 -5586.329,E2 -5586.329} C_VEL
LIN {X 0,Y 509.909,Z 251.776,A -85,B 0,C 180,E1 -5588.72,E2 -5588.72} C_VEL
LIN {X 0,Y 509.943,Z 251.775,A -85,B 0,C 180,E1 -5591.93,E2 -5591.93} C_VEL
LIN {X 0,Y 509.885,Z 251.783,A -85,B 0,C 180,E1 -5595.241,E2 -5595.241} C_VEL
LIN {X 0,Y 509.88,Z 251.783,A -85,B 0,C 180,E1 -5598,E2 -5598} C_VEL
LIN {X 0,Y 509.842,Z 251.786,A -85,B 0,C 180,E1 -5601.001,E2 -5601.001} C_VEL
LIN {X 0,Y 509.861,Z 251.782,A -85,B 0,C 180,E1 -5604.425,E2 -5604.425} C_VEL
LIN {X 0,Y 509.878,Z 251.782,A -85,B 0,C 180,E1 -5607.055,E2 -5607.055} C_VEL
LIN {X 0,Y 509.848,Z 251.79,A -85,B 0,C 180,E1 -5609.751,E2 -5609.751} C_VEL
LIN {X 0,Y 509.868,Z 251.782,A -85,B 0,C 180,E1 -5612.775,E2 -5612.775} C_VEL
LIN {X 0,Y 509.834,Z 251.794,A -85,B 0,C 180,E1 -5615.581,E2 -5615.581} C_VEL
LIN {X 0,Y 509.849,Z 251.784,A -85,B 0,C 180,E1 -5618.337,E2 -5618.337} C_VEL
LIN {X 0,Y 509.85,Z 251.79,A -85,B 0,C 180,E1 -5621.425,E2 -5621.425} C_VEL
LIN {X 0,Y 509.847,Z 251.784,A -85,B 0,C 180,E1 -5624.668,E2 -5624.668} C_VEL
LIN {X 0,Y 509.872,Z 251.783,A -85,B 0,C 180,E1 -5628.1,E2 -5628.1} C_VEL
LIN {X 0,Y 509.85,Z 251.784,A -85,B 0,C 180,E1 -5630.649,E2 -5630.649} C_VEL
LIN {X 0,Y 509.82,Z 251.794,A -85,B 0,C 180,E1 -5633.746,E2 -5633.746} C_VEL
LIN {X 0,Y 509.154,Z 251.872,A -85,B 0,C 180,E1 -5634.406,E2 -5634.406} C_VEL
LIN {X 0,Y 506.336,Z 252.228,A -85,B 0,C 180,E1 -5635.477,E2 -5635.477} C_VEL
LIN {X 0,Y 503.944,Z 252.524,A -85,B 0,C 180,E1 -5636.341,E2 -5636.341} C_VEL
LIN {X 0,Y 502.896,Z 252.652,A -85,B 0,C 180,E1 -5637.007,E2 -5637.007} C_VEL
LIN {X 0,Y 502.799,Z 252.663,A -85,B 0,C 180,E1 -5637.233,E2 -5637.233} C_VEL
LIN {X 0,Y 502.805,Z 252.664,A -85,B 0,C 180,E1 -5640.065,E2 -5640.065} C_VEL
LIN {X 0,Y 502.825,Z 252.659,A -85,B 0,C 180,E1 -5642.533,E2 -5642.533} C_VEL
LIN {X 0,Y 502.822,Z 252.664,A -85,B 0,C 180,E1 -5645.298,E2 -5645.298} C_VEL
LIN {X 0,Y 502.802,Z 252.667,A -85,B 0,C 180,E1 -5647.828,E2 -5647.828} C_VEL
LIN {X 0,Y 502.816,Z 252.66,A -85,B 0,C 180,E1 -5650.4,E2 -5650.4} C_VEL
LIN {X 0,Y 502.826,Z 252.66,A -85,B 0,C 180,E1 -5652.932,E2 -5652.932} C_VEL
LIN {X 0,Y 502.836,Z 252.663,A -85,B 0,C 180,E1 -5655.429,E2 -5655.429} C_VEL
LIN {X 0,Y 502.872,Z 252.653,A -85,B 0,C 180,E1 -5658.717,E2 -5658.717} C_VEL
LIN {X 0,Y 502.893,Z 252.654,A -85,B 0,C 180,E1 -5661.967,E2 -5661.967} C_VEL
LIN {X 0,Y 502.923,Z 252.647,A -85,B 0,C 180,E1 -5664.386,E2 -5664.386} C_VEL
LIN {X 0,Y 503.013,Z 252.643,A -85,B 0,C 180,E1 -5667.598,E2 -5667.598} C_VEL
LIN {X 0,Y 503.014,Z 252.639,A -85,B 0,C 180,E1 -5670,E2 -5670} C_VEL
LIN {X 0,Y 503.012,Z 252.636,A -85,B 0,C 180,E1 -5672.402,E2 -5672.402} C_VEL
LIN {X 0,Y 502.918,Z 252.655,A -85,B 0,C 180,E1 -5675.613,E2 -5675.613} C_VEL
LIN {X 0,Y 502.89,Z 252.654,A -85,B 0,C 180,E1 -5678.033,E2 -5678.033} C_VEL
LIN {X 0,Y 502.882,Z 252.656,A -85,B 0,C 180,E1 -5681.283,E2 -5681.283} C_VEL
LIN {X 0,Y 502.832,Z 252.658,A -85,B 0,C 180,E1 -5684.571,E2 -5684.571} C_VEL
LIN {X 0,Y 502.843,Z 252.661,A -85,B 0,C 180,E1 -5687.907,E2 -5687.907} C_VEL
LIN {X 0,Y 502.818,Z 252.66,A -85,B 0,C 180,E1 -5690.536,E2 -5690.536} C_VEL
LIN {X 0,Y 502.775,Z 252.667,A -85,B 0,C 180,E1 -5693.041,E2 -5693.041} C_VEL
LIN {X 0,Y 502.833,Z 252.658,A -85,B 0,C 180,E1 -5696.556,E2 -5696.556} C_VEL
LIN {X 0,Y 502.81,Z 252.665,A -85,B 0,C 180,E1 -5699.288,E2 -5699.288} C_VEL
LIN {X 0,Y 502.753,Z 252.673,A -85,B 0,C 180,E1 -5702.086,E2 -5702.086} C_VEL
LIN {X 0,Y 502.742,Z 252.763,A -85,B 0,C 180,E1 -5703.186,E2 -5703.186} C_VEL
LIN {X 0,Y 502.626,Z 265.378,A -85,B 0,C 180,E1 -5706.21,E2 -5706.21} C_VEL
LIN {X 0,Y 502.628,Z 267.203,A -85,B 0,C 180,E1 -5706.646,E2 -5706.646} C_VEL
LIN {X 0,Y 504.22,Z 277.181,A -85,B 0,C 180,E1 -5706.838,E2 -5706.838} C_VEL
LIN {X 0,Y 503.821,Z 342.535,A -85,B 0,C 180,E1 -5707.804,E2 -5707.804} C_VEL
LIN {X 0,Y 503.664,Z 352.046,A -85,B 0,C 180,E1 -5708.045,E2 -5708.045} C_VEL
LIN {X 0,Y 503.549,Z 362.494,A -85,B 0,C 180,E1 -5708.443,E2 -5708.443} C_VEL
LIN {X 0,Y 503.348,Z 373.76,A -85,B 0,C 180,E1 -5709.053,E2 -5709.053} C_VEL
LIN {X 0,Y 503.194,Z 381.862,A -85,B 0,C 180,E1 -5709.627,E2 -5709.627} C_VEL
LIN {X 0,Y 502.956,Z 390.529,A -85,B 0,C 180,E1 -5710.391,E2 -5710.391} C_VEL
LIN {X 0,Y 502.752,Z 396.881,A -85,B 0,C 180,E1 -5711.071,E2 -5711.071} C_VEL
LIN {X 0,Y 502.639,Z 403.182,A -85,B 0,C 180,E1 -5711.885,E2 -5711.885} C_VEL
LIN {X 0,Y 502.474,Z 408.51,A -85,B 0,C 180,E1 -5712.714,E2 -5712.714} C_VEL
LIN {X 0,Y 502.383,Z 412.954,A -85,B 0,C 180,E1 -5713.55,E2 -5713.55} C_VEL
LIN {X 0,Y 502.309,Z 416.95,A -85,B 0,C 180,E1 -5714.476,E2 -5714.476} C_VEL
LIN {X 0,Y 502.248,Z 419.035,A -85,B 0,C 180,E1 -5715.039,E2 -5715.039} C_VEL
LIN {X 0,Y 502.148,Z 422.102,A -85,B 0,C 180,E1 -5716.15,E2 -5716.15} C_VEL
LIN {X 0,Y 502.132,Z 423.216,A -85,B 0,C 180,E1 -5716.701,E2 -5716.701} C_VEL
LIN {X 0,Y 502.07,Z 424.894,A -85,B 0,C 180,E1 -5717.892,E2 -5717.892} C_VEL
LIN {X 0,Y 502.045,Z 425.433,A -85,B 0,C 180,E1 -5719.105,E2 -5719.105} C_VEL
LIN {X 0,Y 502.044,Z 424.743,A -85,B 0,C 180,E1 -5720.346,E2 -5720.346} C_VEL
LIN {X 0,Y 502.074,Z 424.021,A -85,B 0,C 180,E1 -5720.958,E2 -5720.958} C_VEL
LIN {X 0,Y 502.153,Z 422.067,A -85,B 0,C 180,E1 -5721.99,E2 -5721.99} C_VEL
LIN {X 0,Y 502.269,Z 419.243,A -85,B 0,C 180,E1 -5723.011,E2 -5723.011} C_VEL
LIN {X 0,Y 502.364,Z 414.525,A -85,B 0,C 180,E1 -5724.232,E2 -5724.232} C_VEL
LIN {X 0,Y 502.497,Z 408.878,A -85,B 0,C 180,E1 -5725.336,E2 -5725.336} C_VEL
LIN {X 0,Y 502.632,Z 403.122,A -85,B 0,C 180,E1 -5726.235,E2 -5726.235} C_VEL
LIN {X 0,Y 502.852,Z 395.277,A -85,B 0,C 180,E1 -5727.227,E2 -5727.227} C_VEL
LIN {X 0,Y 503.105,Z 386.751,A -85,B 0,C 180,E1 -5728.076,E2 -5728.076} C_VEL
LIN {X 0,Y 503.345,Z 377.271,A -85,B 0,C 180,E1 -5728.812,E2 -5728.812} C_VEL
LIN {X 0,Y 503.442,Z 369.281,A -85,B 0,C 180,E1 -5729.31,E2 -5729.31} C_VEL
LIN {X 0,Y 503.589,Z 360.806,A -85,B 0,C 180,E1 -5729.726,E2 -5729.726} C_VEL
LIN {X 0,Y 503.74,Z 351.436,A -85,B 0,C 180,E1 -5730.068,E2 -5730.068} C_VEL
LIN {X 0,Y 503.794,Z 342.697,A -85,B 0,C 180,E1 -5730.287,E2 -5730.287} C_VEL
LIN {X 0,Y 504.077,Z 275.308,A -85,B 0,C 180,E1 -5731.291,E2 -5731.291} C_VEL
LIN {X 0,Y 502.607,Z 266.82,A -85,B 0,C 180,E1 -5731.458,E2 -5731.458} C_VEL
LIN {X 0,Y 502.583,Z 252.969,A -85,B 0,C 180,E1 -5734.311,E2 -5734.311} C_VEL
LIN {X 0,Y 502.63,Z 252.692,A -85,B 0,C 180,E1 -5734.425,E2 -5734.425} C_VEL
LIN {X 0,Y 502.791,Z 252.666,A -85,B 0,C 180,E1 -5737.298,E2 -5737.298} C_VEL
LIN {X 0,Y 502.815,Z 252.671,A -85,B 0,C 180,E1 -5740.401,E2 -5740.401} C_VEL
LIN {X 0,Y 502.825,Z 252.663,A -85,B 0,C 180,E1 -5742.932,E2 -5742.932} C_VEL
LIN {X 0,Y 502.834,Z 252.659,A -85,B 0,C 180,E1 -5745.43,E2 -5745.43} C_VEL
LIN {X 0,Y 502.871,Z 252.66,A -85,B 0,C 180,E1 -5748.717,E2 -5748.717} C_VEL
LIN {X 0,Y 502.892,Z 252.654,A -85,B 0,C 180,E1 -5751.967,E2 -5751.967} C_VEL
LIN {X 0,Y 502.938,Z 252.653,A -85,B 0,C 180,E1 -5754.387,E2 -5754.387} C_VEL
LIN {X 0,Y 503.016,Z 252.634,A -85,B 0,C 180,E1 -5757.598,E2 -5757.598} C_VEL
LIN {X 0,Y 503.017,Z 252.638,A -85,B 0,C 180,E1 -5760.001,E2 -5760.001} C_VEL
LIN {X 0,Y 503.016,Z 252.642,A -85,B 0,C 180,E1 -5762.403,E2 -5762.403} C_VEL
LIN {X 0,Y 502.93,Z 252.645,A -85,B 0,C 180,E1 -5765.614,E2 -5765.614} C_VEL
LIN {X 0,Y 502.893,Z 252.652,A -85,B 0,C 180,E1 -5768.034,E2 -5768.034} C_VEL
LIN {X 0,Y 502.868,Z 252.653,A -85,B 0,C 180,E1 -5771.284,E2 -5771.284} C_VEL
LIN {X 0,Y 502.843,Z 252.664,A -85,B 0,C 180,E1 -5774.571,E2 -5774.571} C_VEL
LIN {X 0,Y 502.854,Z 252.655,A -85,B 0,C 180,E1 -5777.908,E2 -5777.908} C_VEL
LIN {X 0,Y 502.821,Z 252.663,A -85,B 0,C 180,E1 -5780.537,E2 -5780.537} C_VEL
LIN {X 0,Y 502.789,Z 252.665,A -85,B 0,C 180,E1 -5783.041,E2 -5783.041} C_VEL
LIN {X 0,Y 502.835,Z 252.655,A -85,B 0,C 180,E1 -5785.676,E2 -5785.676} C_VEL
LIN {X 0,Y 502.836,Z 252.665,A -85,B 0,C 180,E1 -5788.373,E2 -5788.373} C_VEL
LIN {X 0,Y 502.788,Z 252.664,A -85,B 0,C 180,E1 -5791.5,E2 -5791.5} C_VEL
LIN {X 0,Y 502.8,Z 252.667,A -85,B 0,C 180,E1 -5794.446,E2 -5794.446} C_VEL
LIN {X 0,Y 502.776,Z 252.664,A -85,B 0,C 180,E1 -5797.179,E2 -5797.179} C_VEL
LIN {X 0,Y 502.817,Z 252.663,A -85,B 0,C 180,E1 -5800.013,E2 -5800.013} C_VEL
LIN {X 0,Y 502.767,Z 252.666,A -85,B 0,C 180,E1 -5803.232,E2 -5803.232} C_VEL
LIN {X 0,Y 502.786,Z 252.664,A -85,B 0,C 180,E1 -5805.662,E2 -5805.662} C_VEL
LIN {X 0,Y 502.815,Z 252.662,A -85,B 0,C 180,E1 -5809.006,E2 -5809.006} C_VEL
LIN {X 0,Y 502.79,Z 252.666,A -85,B 0,C 180,E1 -5812.047,E2 -5812.047} C_VEL
LIN {X 0,Y 502.805,Z 252.664,A -85,B 0,C 180,E1 -5815.036,E2 -5815.036} C_VEL
LIN {X 0,Y 502.783,Z 252.667,A -85,B 0,C 180,E1 -5817.916,E2 -5817.916} C_VEL
LIN {X 0,Y 502.82,Z 252.668,A -85,B 0,C 180,E1 -5820.713,E2 -5820.713} C_VEL
LIN {X 0,Y 502.862,Z 252.656,A -85,B 0,C 180,E1 -5823.44,E2 -5823.44} C_VEL
LIN {X 0,Y 502.858,Z 252.785,A -85,B 0,C 180,E1 -5826.282,E2 -5826.282} C_VEL
LIN {X 0,Y 503.73,Z 259.334,A -85,B 0,C 180,E1 -5827.439,E2 -5827.439} C_VEL
LIN {X 0,Y 503.397,Z 274.357,A -85,B 0,C 180,E1 -5829.999,E2 -5829.999} C_VEL
LIN {X 0,Y 503.06,Z 293.003,A -85,B 0,C 180,E1 -5833.149,E2 -5833.149} C_VEL
LIN {X 0,Y 502.763,Z 311.487,A -85,B 0,C 180,E1 -5836.253,E2 -5836.253} C_VEL
LIN {X 0,Y 502.652,Z 319.564,A -85,B 0,C 180,E1 -5837.576,E2 -5837.576} C_VEL
LIN {X 0,Y 504.07,Z 333.535,A -85,B 0,C 180,E1 -5837.816,E2 -5837.816} C_VEL
LIN {X 0,Y 503.76,Z 397.406,A -85,B 0,C 180,E1 -5838.763,E2 -5838.763} C_VEL
LIN {X 0,Y 503.562,Z 407.146,A -85,B 0,C 180,E1 -5839.013,E2 -5839.013} C_VEL
LIN {X 0,Y 503.366,Z 418.261,A -85,B 0,C 180,E1 -5839.441,E2 -5839.441} C_VEL
LIN {X 0,Y 503.103,Z 429.141,A -85,B 0,C 180,E1 -5840.046,E2 -5840.046} C_VEL
LIN {X 0,Y 502.947,Z 437.602,A -85,B 0,C 180,E1 -5840.652,E2 -5840.652} C_VEL
LIN {X 0,Y 502.691,Z 445.593,A -85,B 0,C 180,E1 -5841.356,E2 -5841.356} C_VEL
LIN {X 0,Y 502.502,Z 453.065,A -85,B 0,C 180,E1 -5842.163,E2 -5842.163} C_VEL
LIN {X 0,Y 502.393,Z 459.86,A -85,B 0,C 180,E1 -5843.06,E2 -5843.06} C_VEL
LIN {X 0,Y 502.294,Z 466.616,A -85,B 0,C 180,E1 -5844.178,E2 -5844.178} C_VEL
LIN {X 0,Y 502.144,Z 471.299,A -85,B 0,C 180,E1 -5845.183,E2 -5845.183} C_VEL
LIN {X 0,Y 502.187,Z 474.35,A -85,B 0,C 180,E1 -5845.988,E2 -5845.988} C_VEL
LIN {X 0,Y 502.134,Z 476.712,A -85,B 0,C 180,E1 -5846.791,E2 -5846.791} C_VEL
LIN {X 0,Y 502.123,Z 478.494,A -85,B 0,C 180,E1 -5847.594,E2 -5847.594} C_VEL
LIN {X 0,Y 502.035,Z 479.768,A -85,B 0,C 180,E1 -5848.396,E2 -5848.396} C_VEL
LIN {X 0,Y 502,Z 480.565,A -85,B 0,C 180,E1 -5849.198,E2 -5849.198} C_VEL
LIN {X 0,Y 502,Z 480.874,A -85,B 0,C 180,E1 -5850,E2 -5850} C_VEL
LIN {X 0,Y 501.999,Z 480.583,A -85,B 0,C 180,E1 -5850.802,E2 -5850.802} C_VEL
LIN {X 0,Y 502.035,Z 479.798,A -85,B 0,C 180,E1 -5851.605,E2 -5851.605} C_VEL
LIN {X 0,Y 502.123,Z 478.536,A -85,B 0,C 180,E1 -5852.407,E2 -5852.407} C_VEL
LIN {X 0,Y 502.171,Z 475.606,A -85,B 0,C 180,E1 -5853.611,E2 -5853.611} C_VEL
LIN {X 0,Y 502.146,Z 472.926,A -85,B 0,C 180,E1 -5854.415,E2 -5854.415} C_VEL
LIN {X 0,Y 502.259,Z 467.694,A -85,B 0,C 180,E1 -5855.621,E2 -5855.621} C_VEL
LIN {X 0,Y 502.367,Z 461.942,A -85,B 0,C 180,E1 -5856.648,E2 -5856.648} C_VEL
LIN {X 0,Y 502.472,Z 454.945,A -85,B 0,C 180,E1 -5857.636,E2 -5857.636} C_VEL
LIN {X 0,Y 502.678,Z 446.818,A -85,B 0,C 180,E1 -5858.543,E2 -5858.543} C_VEL
LIN {X 0,Y 502.91,Z 439.057,A -85,B 0,C 180,E1 -5859.248,E2 -5859.248} C_VEL
LIN {X 0,Y 503.086,Z 430.893,A -85,B 0,C 180,E1 -5859.854,E2 -5859.854} C_VEL
LIN {X 0,Y 503.249,Z 422.416,A -85,B 0,C 180,E1 -5860.358,E2 -5860.358} C_VEL
LIN {X 0,Y 503.502,Z 412.524,A -85,B 0,C 180,E1 -5860.811,E2 -5860.811} C_VEL
LIN {X 0,Y 503.708,Z 400.375,A -85,B 0,C 180,E1 -5861.188,E2 -5861.188} C_VEL
LIN {X 0,Y 503.886,Z 380.829,A -85,B 0,C 180,E1 -5861.505,E2 -5861.505} C_VEL
LIN {X 0,Y 503.938,Z 331.171,A -85,B 0,C 180,E1 -5862.226,E2 -5862.226} C_VEL
LIN {X 0,Y 502.652,Z 319.789,A -85,B 0,C 180,E1 -5862.438,E2 -5862.438} C_VEL
LIN {X 0,Y 502.975,Z 303.284,A -85,B 0,C 180,E1 -5865.27,E2 -5865.27} C_VEL
LIN {X 0,Y 503.325,Z 286.541,A -85,B 0,C 180,E1 -5868.172,E2 -5868.172} C_VEL
LIN {X 0,Y 503.878,Z 268.919,A -85,B 0,C 180,E1 -5871.262,E2 -5871.262} C_VEL
LIN {X 0,Y 503.967,Z 259.092,A -85,B 0,C 180,E1 -5873.016,E2 -5873.016} C_VEL
LIN {X 0,Y 502.821,Z 252.665,A -85,B 0,C 180,E1 -5874.241,E2 -5874.241} C_VEL
LIN {X 0,Y 502.824,Z 252.667,A -85,B 0,C 180,E1 -5877.467,E2 -5877.467} C_VEL
LIN {X 0,Y 502.809,Z 252.661,A -85,B 0,C 180,E1 -5880.211,E2 -5880.211} C_VEL
LIN {X 0,Y 502.831,Z 252.66,A -85,B 0,C 180,E1 -5883.031,E2 -5883.031} C_VEL
LIN {X 0,Y 502.775,Z 252.668,A -85,B 0,C 180,E1 -5885.95,E2 -5885.95} C_VEL
LIN {X 0,Y 502.799,Z 252.663,A -85,B 0,C 180,E1 -5888.976,E2 -5888.976} C_VEL
LIN {X 0,Y 502.795,Z 252.663,A -85,B 0,C 180,E1 -5892.139,E2 -5892.139} C_VEL
LIN {X 0,Y 502.799,Z 252.67,A -85,B 0,C 180,E1 -5895.468,E2 -5895.468} C_VEL
LIN {X 0,Y 502.819,Z 252.661,A -85,B 0,C 180,E1 -5898.934,E2 -5898.934} C_VEL
LIN {X 0,Y 502.791,Z 252.665,A -85,B 0,C 180,E1 -5902.045,E2 -5902.045} C_VEL
LIN {X 0,Y 502.804,Z 252.663,A -85,B 0,C 180,E1 -5905.034,E2 -5905.034} C_VEL
LIN {X 0,Y 502.779,Z 252.668,A -85,B 0,C 180,E1 -5907.915,E2 -5907.915} C_VEL
LIN {X 0,Y 502.82,Z 252.659,A -85,B 0,C 180,E1 -5910.712,E2 -5910.712} C_VEL
LIN {X 0,Y 502.877,Z 252.659,A -85,B 0,C 180,E1 -5913.434,E2 -5913.434} C_VEL
LIN {X 0,Y 502.787,Z 252.665,A -85,B 0,C 180,E1 -5916.086,E2 -5916.086} C_VEL
LIN {X 0,Y 502.779,Z 252.664,A -85,B 0,C 180,E1 -5918.688,E2 -5918.688} C_VEL
LIN {X 0,Y 502.825,Z 252.663,A -85,B 0,C 180,E1 -5921.248,E2 -5921.248} C_VEL
LIN {X 0,Y 502.817,Z 252.665,A -85,B 0,C 180,E1 -5923.766,E2 -5923.766} C_VEL
LIN {X 0,Y 502.825,Z 252.659,A -85,B 0,C 180,E1 -5926.254,E2 -5926.254} C_VEL
LIN {X 0,Y 502.871,Z 252.653,A -85,B 0,C 180,E1 -5928.716,E2 -5928.716} C_VEL
LIN {X 0,Y 502.896,Z 252.653,A -85,B 0,C 180,E1 -5931.966,E2 -5931.966} C_VEL
LIN {X 0,Y 502.932,Z 252.645,A -85,B 0,C 180,E1 -5934.386,E2 -5934.386} C_VEL
LIN {X 0,Y 503.018,Z 252.643,A -85,B 0,C 180,E1 -5937.597,E2 -5937.597} C_VEL
LIN {X 0,Y 503.02,Z 252.637,A -85,B 0,C 180,E1 -5939.999,E2 -5939.999} C_VEL
LIN {X 0,Y 503.018,Z 252.635,A -85,B 0,C 180,E1 -5942.402,E2 -5942.402} C_VEL
LIN {X 0,Y 502.931,Z 252.654,A -85,B 0,C 180,E1 -5945.613,E2 -5945.613} C_VEL
LIN {X 0,Y 502.894,Z 252.652,A -85,B 0,C 180,E1 -5948.033,E2 -5948.033} C_VEL
LIN {X 0,Y 502.885,Z 252.656,A -85,B 0,C 180,E1 -5951.282,E2 -5951.282} C_VEL
LIN {X 0,Y 502.837,Z 252.657,A -85,B 0,C 180,E1 -5954.57,E2 -5954.57} C_VEL
LIN {X 0,Y 502.854,Z 252.659,A -85,B 0,C 180,E1 -5957.906,E2 -5957.906} C_VEL
LIN {X 0,Y 502.82,Z 252.659,A -85,B 0,C 180,E1 -5960.536,E2 -5960.536} C_VEL
LIN {X 0,Y 502.785,Z 252.666,A -85,B 0,C 180,E1 -5963.04,E2 -5963.04} C_VEL
LIN {X 0,Y 502.833,Z 252.665,A -85,B 0,C 180,E1 -5965.675,E2 -5965.675} C_VEL
LIN {X 0,Y 502.831,Z 252.658,A -85,B 0,C 180,E1 -5968.372,E2 -5968.372} C_VEL
LIN {X 0,Y 502.787,Z 252.671,A -85,B 0,C 180,E1 -5971.499,E2 -5971.499} C_VEL
LIN {X 0,Y 502.798,Z 252.662,A -85,B 0,C 180,E1 -5974.444,E2 -5974.444} C_VEL
LIN {X 0,Y 502.771,Z 252.669,A -85,B 0,C 180,E1 -5977.178,E2 -5977.178} C_VEL
LIN {X 0,Y 502.812,Z 252.663,A -85,B 0,C 180,E1 -5980.012,E2 -5980.012} C_VEL
LIN {X 0,Y 502.793,Z 252.664,A -85,B 0,C 180,E1 -5982.199,E2 -5982.199} C_VEL
LIN {X 0,Y 502.791,Z 252.67,A -85,B 0,C 180,E1 -5985.468,E2 -5985.468} C_VEL
LIN {X 0,Y 502.826,Z 252.663,A -85,B 0,C 180,E1 -5987.865,E2 -5987.865} C_VEL
LIN {X 0,Y 502.8,Z 252.664,A -85,B 0,C 180,E1 -5991.025,E2 -5991.025} C_VEL
LIN {X 0,Y 502.773,Z 252.667,A -85,B 0,C 180,E1 -5994.167,E2 -5994.167} C_VEL
LIN {X 0,Y 502.799,Z 252.663,A -85,B 0,C 180,E1 -5997.233,E2 -5997.233} C_VEL
LIN {X 0,Y 502.099,Z 252.754,A -85,B 0,C 180,E1 -5997.902,E2 -5997.902} C_VEL
LIN {X 0,Y 499.234,Z 253.108,A -85,B 0,C 180,E1 -5998.987,E2 -5998.987} C_VEL
LIN {X 0,Y 496.838,Z 253.409,A -85,B 0,C 180,E1 -5999.862,E2 -5999.862} C_VEL
LIN {X 0,Y 495.821,Z 253.532,A -85,B 0,C 180,E1 -6000.538,E2 -6000.538} C_VEL
LIN {X 0,Y 495.744,Z 253.541,A -85,B 0,C 180,E1 -6000.767,E2 -6000.767} C_VEL
LIN {X 0,Y 495.782,Z 253.54,A -85,B 0,C 180,E1 -6003.932,E2 -6003.932} C_VEL
LIN {X 0,Y 495.756,Z 253.542,A -85,B 0,C 180,E1 -6007.137,E2 -6007.137} C_VEL
LIN {X 0,Y 495.769,Z 253.54,A -85,B 0,C 180,E1 -6010.11,E2 -6010.11} C_VEL
LIN {X 0,Y 495.778,Z 253.537,A -85,B 0,C 180,E1 -6012.681,E2 -6012.681} C_VEL
LIN {X 0,Y 495.781,Z 253.54,A -85,B 0,C 180,E1 -6015.217,E2 -6015.217} C_VEL
LIN {X 0,Y 495.846,Z 253.528,A -85,B 0,C 180,E1 -6018.555,E2 -6018.555} C_VEL
LIN {X 0,Y 495.864,Z 253.531,A -85,B 0,C 180,E1 -6021.852,E2 -6021.852} C_VEL
LIN {X 0,Y 495.879,Z 253.525,A -85,B 0,C 180,E1 -6024.306,E2 -6024.306} C_VEL
LIN {X 0,Y 495.982,Z 253.519,A -85,B 0,C 180,E1 -6027.563,E2 -6027.563} C_VEL
LIN {X 0,Y 495.985,Z 253.514,A -85,B 0,C 180,E1 -6030,E2 -6030} C_VEL
LIN {X 0,Y 495.981,Z 253.512,A -85,B 0,C 180,E1 -6032.436,E2 -6032.436} C_VEL
LIN {X 0,Y 495.875,Z 253.532,A -85,B 0,C 180,E1 -6035.693,E2 -6035.693} C_VEL
LIN {X 0,Y 495.862,Z 253.528,A -85,B 0,C 180,E1 -6038.148,E2 -6038.148} C_VEL
LIN {X 0,Y 495.857,Z 253.533,A -85,B 0,C 180,E1 -6041.445,E2 -6041.445} C_VEL
LIN {X 0,Y 495.778,Z 253.537,A -85,B 0,C 180,E1 -6044.783,E2 -6044.783} C_VEL
LIN {X 0,Y 495.768,Z 253.542,A -85,B 0,C 180,E1 -6047.319,E2 -6047.319} C_VEL
LIN {X 0,Y 495.758,Z 253.544,A -85,B 0,C 180,E1 -6049.89,E2 -6049.89} C_VEL
LIN {X 0,Y 495.747,Z 253.542,A -85,B 0,C 180,E1 -6052.86,E2 -6052.86} C_VEL
LIN {X 0,Y 495.748,Z 253.543,A -85,B 0,C 180,E1 -6056.069,E2 -6056.069} C_VEL
LIN {X 0,Y 495.757,Z 253.54,A -85,B 0,C 180,E1 -6058.815,E2 -6058.815} C_VEL
LIN {X 0,Y 495.734,Z 253.55,A -85,B 0,C 180,E1 -6061.723,E2 -6061.723} C_VEL
LIN {X 0,Y 495.738,Z 253.732,A -85,B 0,C 180,E1 -6063.156,E2 -6063.156} C_VEL
LIN {X 0,Y 495.609,Z 267.392,A -85,B 0,C 180,E1 -6066.437,E2 -6066.437} C_VEL
LIN {X 0,Y 495.709,Z 268.17,A -85,B 0,C 180,E1 -6066.487,E2 -6066.487} C_VEL
LIN {X 0,Y 497.255,Z 277.324,A -85,B 0,C 180,E1 -6066.664,E2 -6066.664} C_VEL
LIN {X 0,Y 496.876,Z 342.914,A -85,B 0,C 180,E1 -6067.652,E2 -6067.652} C_VEL
LIN {X 0,Y 496.68,Z 352.765,A -85,B 0,C 180,E1 -6067.907,E2 -6067.907} C_VEL
LIN {X 0,Y 496.589,Z 363.637,A -85,B 0,C 180,E1 -6068.333,E2 -6068.333} C_VEL
LIN {X 0,Y 496.359,Z 374.717,A -85,B 0,C 180,E1 -6068.958,E2 -6068.958} C_VEL
LIN {X 0,Y 496.175,Z 383.404,A -85,B 0,C 180,E1 -6069.597,E2 -6069.597} C_VEL
LIN {X 0,Y 495.962,Z 390.075,A -85,B 0,C 180,E1 -6070.191,E2 -6070.191} C_VEL
LIN {X 0,Y 495.733,Z 397.486,A -85,B 0,C 180,E1 -6070.991,E2 -6070.991} C_VEL
LIN {X 0,Y 495.569,Z 404.774,A -85,B 0,C 180,E1 -6071.963,E2 -6071.963} C_VEL
LIN {X 0,Y 495.387,Z 410.558,A -85,B 0,C 180,E1 -6072.918,E2 -6072.918} C_VEL
LIN {X 0,Y 495.262,Z 415.98,A -85,B 0,C 180,E1 -6074.052,E2 -6074.052} C_VEL
LIN {X 0,Y 495.137,Z 420.071,A -85,B 0,C 180,E1 -6075.209,E2 -6075.209} C_VEL
LIN {X 0,Y 495.059,Z 423.035,A -85,B 0,C 180,E1 -6076.385,E2 -6076.385} C_VEL
LIN {X 0,Y 495.018,Z 424.282,A -85,B 0,C 180,E1 -6077.042,E2 -6077.042} C_VEL
LIN {X 0,Y 494.979,Z 425.486,A -85,B 0,C 180,E1 -6078.14,E2 -6078.14} C_VEL
LIN {X 0,Y 494.951,Z 425.789,A -85,B 0,C 180,E1 -6079.22,E2 -6079.22} C_VEL
LIN {X 0,Y 494.98,Z 425.224,A -85,B 0,C 180,E1 -6080.289,E2 -6080.289} C_VEL
LIN {X 0,Y 495.03,Z 423.817,A -85,B 0,C 180,E1 -6081.343,E2 -6081.343} C_VEL
LIN {X 0,Y 495.143,Z 420.845,A -85,B 0,C 180,E1 -6082.64,E2 -6082.64} C_VEL
LIN {X 0,Y 495.242,Z 417.26,A -85,B 0,C 180,E1 -6083.728,E2 -6083.728} C_VEL
LIN {X 0,Y 495.394,Z 412.017,A -85,B 0,C 180,E1 -6084.929,E2 -6084.929} C_VEL
LIN {X 0,Y 495.547,Z 406.31,A -85,B 0,C 180,E1 -6085.932,E2 -6085.932} C_VEL
LIN {X 0,Y 495.733,Z 398.746,A -85,B 0,C 180,E1 -6086.972,E2 -6086.972} C_VEL
LIN {X 0,Y 495.982,Z 391.843,A -85,B 0,C 180,E1 -6087.744,E2 -6087.744} C_VEL
LIN {X 0,Y 496.163,Z 384.858,A -85,B 0,C 180,E1 -6088.394,E2 -6088.394} C_VEL
LIN {X 0,Y 496.379,Z 376.883,A -85,B 0,C 180,E1 -6089.003,E2 -6089.003} C_VEL
LIN {X 0,Y 496.493,Z 369.46,A -85,B 0,C 180,E1 -6089.465,E2 -6089.465} C_VEL
LIN {X 0,Y 496.637,Z 360.427,A -85,B 0,C 180,E1 -6089.908,E2 -6089.908} C_VEL
LIN {X 0,Y 496.787,Z 351.053,A -85,B 0,C 180,E1 -6090.246,E2 -6090.246} C_VEL
LIN {X 0,Y 496.882,Z 340.873,A -85,B 0,C 180,E1 -6090.489,E2 -6090.489} C_VEL
LIN {X 0,Y 497.241,Z 276.509,A -85,B 0,C 180,E1 -6091.45,E2 -6091.45} C_VEL
LIN {X 0,Y 495.619,Z 267.213,A -85,B 0,C 180,E1 -6091.634,E2 -6091.634} C_VEL
LIN {X 0,Y 495.591,Z 253.569,A -85,B 0,C 180,E1 -6094.458,E2 -6094.458} C_VEL
LIN {X 0,Y 495.746,Z 253.545,A -85,B 0,C 180,E1 -6097.14,E2 -6097.14} C_VEL
LIN {X 0,Y 495.767,Z 253.546,A -85,B 0,C 180,E1 -6100.11,E2 -6100.11} C_VEL
LIN {X 0,Y 495.777,Z 253.544,A -85,B 0,C 180,E1 -6102.682,E2 -6102.682} C_VEL
LIN {X 0,Y 495.779,Z 253.538,A -85,B 0,C 180,E1 -6105.218,E2 -6105.218} C_VEL
LIN {X 0,Y 495.844,Z 253.538,A -85,B 0,C 180,E1 -6108.555,E2 -6108.555} C_VEL
LIN {X 0,Y 495.863,Z 253.528,A -85,B 0,C 180,E1 -6111.853,E2 -6111.853} C_VEL
LIN {X 0,Y 495.894,Z 253.529,A -85,B 0,C 180,E1 -6114.307,E2 -6114.307} C_VEL
LIN {X 0,Y 495.984,Z 253.51,A -85,B 0,C 180,E1 -6117.564,E2 -6117.564} C_VEL
LIN {X 0,Y 495.988,Z 253.513,A -85,B 0,C 180,E1 -6120.001,E2 -6120.001} C_VEL
LIN {X 0,Y 495.985,Z 253.518,A -85,B 0,C 180,E1 -6122.437,E2 -6122.437} C_VEL
LIN {X 0,Y 495.888,Z 253.523,A -85,B 0,C 180,E1 -6125.694,E2 -6125.694} C_VEL
LIN {X 0,Y 495.865,Z 253.529,A -85,B 0,C 180,E1 -6128.149,E2 -6128.149} C_VEL
LIN {X 0,Y 495.843,Z 253.528,A -85,B 0,C 180,E1 -6131.446,E2 -6131.446} C_VEL
LIN {X 0,Y 495.786,Z 253.54,A -85,B 0,C 180,E1 -6134.784,E2 -6134.784} C_VEL
LIN {X 0,Y 495.78,Z 253.535,A -85,B 0,C 180,E1 -6137.319,E2 -6137.319} C_VEL
LIN {X 0,Y 495.77,Z 253.538,A -85,B 0,C 180,E1 -6139.891,E2 -6139.891} C_VEL
LIN {X 0,Y 495.751,Z 253.543,A -85,B 0,C 180,E1 -6142.861,E2 -6142.861} C_VEL
LIN {X 0,Y 495.792,Z 253.535,A -85,B 0,C 180,E1 -6146.068,E2 -6146.068} C_VEL
LIN {X 0,Y 495.774,Z 253.538,A -85,B 0,C 180,E1 -6148.815,E2 -6148.815} C_VEL
LIN {X 0,Y 495.75,Z 253.541,A -85,B 0,C 180,E1 -6151.726,E2 -6151.726} C_VEL
LIN {X 0,Y 495.77,Z 253.544,A -85,B 0,C 180,E1 -6154.696,E2 -6154.696} C_VEL
LIN {X 0,Y 495.727,Z 253.541,A -85,B 0,C 180,E1 -6157.562,E2 -6157.562} C_VEL
LIN {X 0,Y 495.775,Z 253.542,A -85,B 0,C 180,E1 -6160.699,E2 -6160.699} C_VEL
LIN {X 0,Y 495.729,Z 253.544,A -85,B 0,C 180,E1 -6164.002,E2 -6164.002} C_VEL
LIN {X 0,Y 495.722,Z 253.545,A -85,B 0,C 180,E1 -6167.118,E2 -6167.118} C_VEL
LIN {X 0,Y 495.755,Z 253.542,A -85,B 0,C 180,E1 -6169.954,E2 -6169.954} C_VEL
LIN {X 0,Y 495.727,Z 253.551,A -85,B 0,C 180,E1 -6172.554,E2 -6172.554} C_VEL
LIN {X 0,Y 495.781,Z 253.537,A -85,B 0,C 180,E1 -6175.458,E2 -6175.458} C_VEL
LIN {X 0,Y 495.754,Z 253.547,A -85,B 0,C 180,E1 -6178.365,E2 -6178.365} C_VEL
LIN {X 0,Y 495.784,Z 253.539,A -85,B 0,C 180,E1 -6181.508,E2 -6181.508} C_VEL
LIN {X 0,Y 495.778,Z 253.541,A -85,B 0,C 180,E1 -6183.932,E2 -6183.932} C_VEL
LIN {X 0,Y 495.801,Z 253.684,A -85,B 0,C 180,E1 -6186.173,E2 -6186.173} C_VEL
LIN {X 0,Y 496.71,Z 259.616,A -85,B 0,C 180,E1 -6187.242,E2 -6187.242} C_VEL
LIN {X 0,Y 496.405,Z 273.848,A -85,B 0,C 180,E1 -6189.705,E2 -6189.705} C_VEL
LIN {X 0,Y 496.064,Z 291.292,A -85,B 0,C 180,E1 -6192.692,E2 -6192.692} C_VEL
LIN {X 0,Y 495.712,Z 311.047,A -85,B 0,C 180,E1 -6196.054,E2 -6196.054} C_VEL
LIN {X 0,Y 495.58,Z 318.814,A -85,B 0,C 180,E1 -6197.373,E2 -6197.373} C_VEL
LIN {X 0,Y 497.137,Z 335.143,A -85,B 0,C 180,E1 -6197.672,E2 -6197.672} C_VEL
LIN {X 0,Y 496.796,Z 396.876,A -85,B 0,C 180,E1 -6198.603,E2 -6198.603} C_VEL
LIN {X 0,Y 496.6,Z 406.645,A -85,B 0,C 180,E1 -6198.857,E2 -6198.857} C_VEL
LIN {X 0,Y 496.364,Z 417.777,A -85,B 0,C 180,E1 -6199.291,E2 -6199.291} C_VEL
LIN {X 0,Y 496.096,Z 428.678,A -85,B 0,C 180,E1 -6199.904,E2 -6199.904} C_VEL
LIN {X 0,Y 495.918,Z 437.146,A -85,B 0,C 180,E1 -6200.518,E2 -6200.518} C_VEL
LIN {X 0,Y 495.701,Z 444.116,A -85,B 0,C 180,E1 -6201.131,E2 -6201.131} C_VEL
LIN {X 0,Y 495.475,Z 450.9,A -85,B 0,C 180,E1 -6201.846,E2 -6201.846} C_VEL
LIN {X 0,Y 495.372,Z 457.344,A -85,B 0,C 180,E1 -6202.664,E2 -6202.664} C_VEL
LIN {X 0,Y 495.251,Z 462.7,A -85,B 0,C 180,E1 -6203.482,E2 -6203.482} C_VEL
LIN {X 0,Y 495.187,Z 467.17,A -85,B 0,C 180,E1 -6204.299,E2 -6204.299} C_VEL
LIN {X 0,Y 495.049,Z 472.433,A -85,B 0,C 180,E1 -6205.522,E2 -6205.522} C_VEL
LIN {X 0,Y 495.095,Z 475.136,A -85,B 0,C 180,E1 -6206.338,E2 -6206.338} C_VEL
LIN {X 0,Y 495.056,Z 478.097,A -85,B 0,C 180,E1 -6207.559,E2 -6207.559} C_VEL
LIN {X 0,Y 494.962,Z 479.375,A -85,B 0,C 180,E1 -6208.373,E2 -6208.373} C_VEL
LIN {X 0,Y 494.919,Z 480.173,A -85,B 0,C 180,E1 -6209.187,E2 -6209.187} C_VEL
LIN {X 0,Y 494.916,Z 480.483,A -85,B 0,C 180,E1 -6210,E2 -6210} C_VEL
LIN {X 0,Y 494.919,Z 480.193,A -85,B 0,C 180,E1 -6210.814,E2 -6210.814} C_VEL
LIN {X 0,Y 494.962,Z 479.409,A -85,B 0,C 180,E1 -6211.627,E2 -6211.627} C_VEL
LIN {X 0,Y 495.056,Z 478.147,A -85,B 0,C 180,E1 -6212.441,E2 -6212.441} C_VEL
LIN {X 0,Y 495.095,Z 475.214,A -85,B 0,C 180,E1 -6213.663,E2 -6213.663} C_VEL
LIN {X 0,Y 495.048,Z 472.529,A -85,B 0,C 180,E1 -6214.478,E2 -6214.478} C_VEL
LIN {X 0,Y 495.187,Z 467.295,A -85,B 0,C 180,E1 -6215.702,E2 -6215.702} C_VEL
LIN {X 0,Y 495.291,Z 460.646,A -85,B 0,C 180,E1 -6216.887,E2 -6216.887} C_VEL
LIN {X 0,Y 495.431,Z 452.814,A -85,B 0,C 180,E1 -6217.95,E2 -6217.95} C_VEL
LIN {X 0,Y 495.674,Z 445.366,A -85,B 0,C 180,E1 -6218.767,E2 -6218.767} C_VEL
LIN {X 0,Y 495.933,Z 437.387,A -85,B 0,C 180,E1 -6219.482,E2 -6219.482} C_VEL
LIN {X 0,Y 496.17,Z 427.428,A -85,B 0,C 180,E1 -6220.198,E2 -6220.198} C_VEL
LIN {X 0,Y 496.424,Z 416.873,A -85,B 0,C 180,E1 -6220.76,E2 -6220.76} C_VEL
LIN {X 0,Y 496.595,Z 406.945,A -85,B 0,C 180,E1 -6221.144,E2 -6221.144} C_VEL
LIN {X 0,Y 496.792,Z 397.18,A -85,B 0,C 180,E1 -6221.397,E2 -6221.397} C_VEL
LIN {X 0,Y 497.06,Z 332.377,A -85,B 0,C 180,E1 -6222.374,E2 -6222.374} C_VEL
LIN {X 0,Y 495.606,Z 319.501,A -85,B 0,C 180,E1 -6222.604,E2 -6222.604} C_VEL
LIN {X 0,Y 495.989,Z 302.2,A -85,B 0,C 180,E1 -6225.618,E2 -6225.618} C_VEL
LIN {X 0,Y 496.401,Z 284.95,A -85,B 0,C 180,E1 -6228.657,E2 -6228.657} C_VEL
LIN {X 0,Y 496.933,Z 267.351,A -85,B 0,C 180,E1 -6231.792,E2 -6231.792} C_VEL
LIN {X 0,Y 496.94,Z 259.722,A -85,B 0,C 180,E1 -6233.181,E2 -6233.181} C_VEL
LIN {X 0,Y 495.776,Z 253.542,A -85,B 0,C 180,E1 -6234.405,E2 -6234.405} C_VEL
LIN {X 0,Y 495.783,Z 253.54,A -85,B 0,C 180,E1 -6236.976,E2 -6236.976} C_VEL
LIN {X 0,Y 495.766,Z 253.543,A -85,B 0,C 180,E1 -6239.746,E2 -6239.746} C_VEL
LIN {X 0,Y 495.767,Z 253.537,A -85,B 0,C 180,E1 -6242.594,E2 -6242.594} C_VEL
LIN {X 0,Y 495.75,Z 253.549,A -85,B 0,C 180,E1 -6245.537,E2 -6245.537} C_VEL
LIN {X 0,Y 495.761,Z 253.539,A -85,B 0,C 180,E1 -6248.767,E2 -6248.767} C_VEL
LIN {X 0,Y 495.755,Z 253.544,A -85,B 0,C 180,E1 -6251.78,E2 -6251.78} C_VEL
LIN {X 0,Y 495.748,Z 253.543,A -85,B 0,C 180,E1 -6255.139,E2 -6255.139} C_VEL
LIN {X 0,Y 495.755,Z 253.54,A -85,B 0,C 180,E1 -6258.218,E2 -6258.218} C_VEL
LIN {X 0,Y 495.748,Z 253.547,A -85,B 0,C 180,E1 -6261.408,E2 -6261.408} C_VEL
LIN {X 0,Y 495.752,Z 253.539,A -85,B 0,C 180,E1 -6264.462,E2 -6264.462} C_VEL
LIN {X 0,Y 495.764,Z 253.545,A -85,B 0,C 180,E1 -6267.405,E2 -6267.405} C_VEL
LIN {X 0,Y 495.762,Z 253.539,A -85,B 0,C 180,E1 -6270.253,E2 -6270.253} C_VEL
LIN {X 0,Y 495.83,Z 253.534,A -85,B 0,C 180,E1 -6273.248,E2 -6273.248} C_VEL
LIN {X 0,Y 495.749,Z 253.546,A -85,B 0,C 180,E1 -6275.724,E2 -6275.724} C_VEL
LIN {X 0,Y 495.739,Z 253.541,A -85,B 0,C 180,E1 -6278.37,E2 -6278.37} C_VEL
LIN {X 0,Y 495.779,Z 253.538,A -85,B 0,C 180,E1 -6280.971,E2 -6280.971} C_VEL
LIN {X 0,Y 495.774,Z 253.545,A -85,B 0,C 180,E1 -6283.529,E2 -6283.529} C_VEL
LIN {X 0,Y 495.788,Z 253.537,A -85,B 0,C 180,E1 -6286.055,E2 -6286.055} C_VEL
LIN {X 0,Y 495.846,Z 253.528,A -85,B 0,C 180,E1 -6288.554,E2 -6288.554} C_VEL
LIN {X 0,Y 495.868,Z 253.53,A -85,B 0,C 180,E1 -6291.851,E2 -6291.851} C_VEL
LIN {X 0,Y 495.89,Z 253.523,A -85,B 0,C 180,E1 -6294.306,E2 -6294.306} C_VEL
LIN {X 0,Y 495.987,Z 253.519,A -85,B 0,C 180,E1 -6297.563,E2 -6297.563} C_VEL
LIN {X 0,Y 495.991,Z 253.513,A -85,B 0,C 180,E1 -6299.999,E2 -6299.999} C_VEL
LIN {X 0,Y 495.987,Z 253.51,A -85,B 0,C 180,E1 -6302.436,E2 -6302.436} C_VEL
LIN {X 0,Y 495.889,Z 253.529,A -85,B 0,C 180,E1 -6305.693,E2 -6305.693} C_VEL
LIN {X 0,Y 495.866,Z 253.527,A -85,B 0,C 180,E1 -6308.147,E2 -6308.147} C_VEL
LIN {X 0,Y 495.86,Z 253.533,A -85,B 0,C 180,E1 -6311.444,E2 -6311.444} C_VEL
LIN {X 0,Y 495.782,Z 253.537,A -85,B 0,C 180,E1 -6314.782,E2 -6314.782} C_VEL
LIN {X 0,Y 495.78,Z 253.541,A -85,B 0,C 180,E1 -6317.318,E2 -6317.318} C_VEL
LIN {X 0,Y 495.77,Z 253.542,A -85,B 0,C 180,E1 -6319.889,E2 -6319.889} C_VEL
LIN {X 0,Y 495.752,Z 253.541,A -85,B 0,C 180,E1 -6322.861,E2 -6322.861} C_VEL
LIN {X 0,Y 495.79,Z 253.537,A -85,B 0,C 180,E1 -6326.067,E2 -6326.067} C_VEL
LIN {X 0,Y 495.763,Z 253.539,A -85,B 0,C 180,E1 -6328.814,E2 -6328.814} C_VEL
LIN {X 0,Y 495.75,Z 253.547,A -85,B 0,C 180,E1 -6331.726,E2 -6331.726} C_VEL
LIN {X 0,Y 495.768,Z 253.538,A -85,B 0,C 180,E1 -6334.695,E2 -6334.695} C_VEL
LIN {X 0,Y 495.724,Z 253.551,A -85,B 0,C 180,E1 -6337.561,E2 -6337.561} C_VEL
LIN {X 0,Y 495.779,Z 253.539,A -85,B 0,C 180,E1 -6340.051,E2 -6340.051} C_VEL
LIN {X 0,Y 495.724,Z 253.544,A -85,B 0,C 180,E1 -6342.882,E2 -6342.882} C_VEL
LIN {X 0,Y 495.727,Z 253.546,A -85,B 0,C 180,E1 -6345.999,E2 -6345.999} C_VEL
LIN {X 0,Y 495.759,Z 253.539,A -85,B 0,C 180,E1 -6348.705,E2 -6348.705} C_VEL
LIN {X 0,Y 495.745,Z 253.546,A -85,B 0,C 180,E1 -6351.409,E2 -6351.409} C_VEL
LIN {X 0,Y 495.746,Z 253.541,A -85,B 0,C 180,E1 -6354.463,E2 -6354.463} C_VEL
LIN {X 0,Y 495.76,Z 253.545,A -85,B 0,C 180,E1 -6357.406,E2 -6357.406} C_VEL
LIN {X 0,Y 495.757,Z 253.54,A -85,B 0,C 180,E1 -6360.253,E2 -6360.253} C_VEL
LIN {X 0,Y 495.744,Z 253.541,A -85,B 0,C 180,E1 -6360.767,E2 -6360.767} C_VEL
LIN {X 0,Y 495.087,Z 253.629,A -85,B 0,C 180,E1 -6361.446,E2 -6361.446} C_VEL
LIN {X 0,Y 492.231,Z 253.981,A -85,B 0,C 180,E1 -6362.548,E2 -6362.548} C_VEL
LIN {X 0,Y 489.822,Z 254.285,A -85,B 0,C 180,E1 -6363.437,E2 -6363.437} C_VEL
LIN {X 0,Y 488.806,Z 254.407,A -85,B 0,C 180,E1 -6364.123,E2 -6364.123} C_VEL
LIN {X 0,Y 488.734,Z 254.414,A -85,B 0,C 180,E1 -6364.356,E2 -6364.356} C_VEL
LIN {X 0,Y 488.718,Z 254.419,A -85,B 0,C 180,E1 -6367.153,E2 -6367.153} C_VEL
LIN {X 0,Y 488.72,Z 254.422,A -85,B 0,C 180,E1 -6369.81,E2 -6369.81} C_VEL
LIN {X 0,Y 488.725,Z 254.416,A -85,B 0,C 180,E1 -6372.423,E2 -6372.423} C_VEL
LIN {X 0,Y 488.753,Z 254.414,A -85,B 0,C 180,E1 -6374.999,E2 -6374.999} C_VEL
LIN {X 0,Y 488.799,Z 254.407,A -85,B 0,C 180,E1 -6378.387,E2 -6378.387} C_VEL
LIN {X 0,Y 488.809,Z 254.412,A -85,B 0,C 180,E1 -6381.733,E2 -6381.733} C_VEL
LIN {X 0,Y 488.837,Z 254.403,A -85,B 0,C 180,E1 -6384.224,E2 -6384.224} C_VEL
LIN {X 0,Y 488.95,Z 254.394,A -85,B 0,C 180,E1 -6387.528,E2 -6387.528} C_VEL
LIN {X 0,Y 488.957,Z 254.39,A -85,B 0,C 180,E1 -6390,E2 -6390} C_VEL
LIN {X 0,Y 488.949,Z 254.388,A -85,B 0,C 180,E1 -6392.471,E2 -6392.471} C_VEL
LIN {X 0,Y 488.833,Z 254.408,A -85,B 0,C 180,E1 -6395.776,E2 -6395.776} C_VEL
LIN {X 0,Y 488.806,Z 254.407,A -85,B 0,C 180,E1 -6398.266,E2 -6398.266} C_VEL
LIN {X 0,Y 488.819,Z 254.411,A -85,B 0,C 180,E1 -6401.612,E2 -6401.612} C_VEL
LIN {X 0,Y 488.75,Z 254.414,A -85,B 0,C 180,E1 -6405,E2 -6405} C_VEL
LIN {X 0,Y 488.744,Z 254.414,A -85,B 0,C 180,E1 -6408.442,E2 -6408.442} C_VEL
LIN {X 0,Y 488.696,Z 254.422,A -85,B 0,C 180,E1 -6411.071,E2 -6411.071} C_VEL
LIN {X 0,Y 488.661,Z 254.43,A -85,B 0,C 180,E1 -6413.746,E2 -6413.746} C_VEL
LIN {X 0,Y 488.736,Z 254.416,A -85,B 0,C 180,E1 -6416.933,E2 -6416.933} C_VEL
LIN {X 0,Y 488.71,Z 254.421,A -85,B 0,C 180,E1 -6419.27,E2 -6419.27} C_VEL
LIN {X 0,Y 488.678,Z 254.425,A -85,B 0,C 180,E1 -6422.636,E2 -6422.636} C_VEL
LIN {X 0,Y 488.708,Z 254.454,A -85,B 0,C 180,E1 -6423.063,E2 -6423.063} C_VEL
LIN {X 0,Y 488.584,Z 266.128,A -85,B 0,C 180,E1 -6425.884,E2 -6425.884} C_VEL
LIN {X 0,Y 488.589,Z 267.831,A -85,B 0,C 180,E1 -6426.293,E2 -6426.293} C_VEL
LIN {X 0,Y 490.27,Z 277.553,A -85,B 0,C 180,E1 -6426.488,E2 -6426.488} C_VEL
LIN {X 0,Y 489.907,Z 343.583,A -85,B 0,C 180,E1 -6427.501,E2 -6427.501} C_VEL
LIN {X 0,Y 489.733,Z 353.822,A -85,B 0,C 180,E1 -6427.776,E2 -6427.776} C_VEL
LIN {X 0,Y 489.619,Z 365.176,A -85,B 0,C 180,E1 -6428.243,E2 -6428.243} C_VEL
LIN {X 0,Y 489.369,Z 374.686,A -85,B 0,C 180,E1 -6428.792,E2 -6428.792} C_VEL
LIN {X 0,Y 489.173,Z 383.85,A -85,B 0,C 180,E1 -6429.474,E2 -6429.474} C_VEL
LIN {X 0,Y 488.933,Z 391.404,A -85,B 0,C 180,E1 -6430.167,E2 -6430.167} C_VEL
LIN {X 0,Y 488.712,Z 397.734,A -85,B 0,C 180,E1 -6430.866,E2 -6430.866} C_VEL
LIN {X 0,Y 488.567,Z 403.211,A -85,B 0,C 180,E1 -6431.583,E2 -6431.583} C_VEL
LIN {X 0,Y 488.367,Z 409.37,A -85,B 0,C 180,E1 -6432.559,E2 -6432.559} C_VEL
LIN {X 0,Y 488.251,Z 413.979,A -85,B 0,C 180,E1 -6433.457,E2 -6433.457} C_VEL
LIN {X 0,Y 488.158,Z 418.08,A -85,B 0,C 180,E1 -6434.452,E2 -6434.452} C_VEL
LIN {X 0,Y 488.062,Z 420.36,A -85,B 0,C 180,E1 -6435.124,E2 -6435.124} C_VEL
LIN {X 0,Y 487.986,Z 423.259,A -85,B 0,C 180,E1 -6436.269,E2 -6436.269} C_VEL
LIN {X 0,Y 487.917,Z 425.116,A -85,B 0,C 180,E1 -6437.392,E2 -6437.392} C_VEL
LIN {X 0,Y 487.881,Z 426.029,A -85,B 0,C 180,E1 -6438.508,E2 -6438.508} C_VEL
LIN {X 0,Y 487.869,Z 425.979,A -85,B 0,C 180,E1 -6439.771,E2 -6439.771} C_VEL
LIN {X 0,Y 487.918,Z 424.757,A -85,B 0,C 180,E1 -6441.06,E2 -6441.06} C_VEL
LIN {X 0,Y 488.036,Z 422.123,A -85,B 0,C 180,E1 -6442.374,E2 -6442.374} C_VEL
LIN {X 0,Y 488.13,Z 419.499,A -85,B 0,C 180,E1 -6443.291,E2 -6443.291} C_VEL
LIN {X 0,Y 488.239,Z 415.506,A -85,B 0,C 180,E1 -6444.341,E2 -6444.341} C_VEL
LIN {X 0,Y 488.392,Z 410.896,A -85,B 0,C 180,E1 -6445.299,E2 -6445.299} C_VEL
LIN {X 0,Y 488.531,Z 405.3,A -85,B 0,C 180,E1 -6446.239,E2 -6446.239} C_VEL
LIN {X 0,Y 488.724,Z 398.84,A -85,B 0,C 180,E1 -6447.123,E2 -6447.123} C_VEL
LIN {X 0,Y 488.973,Z 392.188,A -85,B 0,C 180,E1 -6447.874,E2 -6447.874} C_VEL
LIN {X 0,Y 489.154,Z 385.662,A -85,B 0,C 180,E1 -6448.493,E2 -6448.493} C_VEL
LIN {X 0,Y 489.408,Z 377.475,A -85,B 0,C 180,E1 -6449.13,E2 -6449.13} C_VEL
LIN {X 0,Y 489.521,Z 369.508,A -85,B 0,C 180,E1 -6449.633,E2 -6449.633} C_VEL
LIN {X 0,Y 489.717,Z 360.239,A -85,B 0,C 180,E1 -6450.087,E2 -6450.087} C_VEL
LIN {X 0,Y 489.855,Z 349.532,A -85,B 0,C 180,E1 -6450.466,E2 -6450.466} C_VEL
LIN {X 0,Y 489.969,Z 334.981,A -85,B 0,C 180,E1 -6450.754,E2 -6450.754} C_VEL
LIN {X 0,Y 490.322,Z 277.18,A -85,B 0,C 180,E1 -6451.624,E2 -6451.624} C_VEL
LIN {X 0,Y 488.614,Z 267.459,A -85,B 0,C 180,E1 -6451.839,E2 -6451.839} C_VEL
LIN {X 0,Y 488.589,Z 254.441,A -85,B 0,C 180,E1 -6454.552,E2 -6454.552} C_VEL
LIN {X 0,Y 488.709,Z 254.422,A -85,B 0,C 180,E1 -6457.153,E2 -6457.153} C_VEL
LIN {X 0,Y 488.717,Z 254.422,A -85,B 0,C 180,E1 -6459.811,E2 -6459.811} C_VEL
LIN {X 0,Y 488.724,Z 254.425,A -85,B 0,C 180,E1 -6462.424,E2 -6462.424} C_VEL
LIN {X 0,Y 488.751,Z 254.415,A -85,B 0,C 180,E1 -6465,E2 -6465} C_VEL
LIN {X 0,Y 488.797,Z 254.413,A -85,B 0,C 180,E1 -6468.388,E2 -6468.388} C_VEL
LIN {X 0,Y 488.808,Z 254.407,A -85,B 0,C 180,E1 -6471.734,E2 -6471.734} C_VEL
LIN {X 0,Y 488.852,Z 254.405,A -85,B 0,C 180,E1 -6474.225,E2 -6474.225} C_VEL
LIN {X 0,Y 488.952,Z 254.386,A -85,B 0,C 180,E1 -6477.529,E2 -6477.529} C_VEL
LIN {X 0,Y 488.967,Z 254.388,A -85,B 0,C 180,E1 -6480.824,E2 -6480.824} C_VEL
LIN {X 0,Y 488.953,Z 254.394,A -85,B 0,C 180,E1 -6482.472,E2 -6482.472} C_VEL
LIN {X 0,Y 488.847,Z 254.4,A -85,B 0,C 180,E1 -6485.776,E2 -6485.776} C_VEL
LIN {X 0,Y 488.809,Z 254.409,A -85,B 0,C 180,E1 -6488.267,E2 -6488.267} C_VEL
LIN {X 0,Y 488.796,Z 254.406,A -85,B 0,C 180,E1 -6491.613,E2 -6491.613} C_VEL
LIN {X 0,Y 488.756,Z 254.413,A -85,B 0,C 180,E1 -6495.001,E2 -6495.001} C_VEL
LIN {X 0,Y 488.747,Z 254.419,A -85,B 0,C 180,E1 -6498.443,E2 -6498.443} C_VEL
LIN {X 0,Y 488.7,Z 254.417,A -85,B 0,C 180,E1 -6501.072,E2 -6501.072} C_VEL
LIN {X 0,Y 488.686,Z 254.42,A -85,B 0,C 180,E1 -6503.746,E2 -6503.746} C_VEL
LIN {X 0,Y 488.792,Z 254.41,A -85,B 0,C 180,E1 -6506.946,E2 -6506.946} C_VEL
LIN {X 0,Y 488.712,Z 254.42,A -85,B 0,C 180,E1 -6510.366,E2 -6510.366} C_VEL
LIN {X 0,Y 488.73,Z 254.411,A -85,B 0,C 180,E1 -6513.485,E2 -6513.485} C_VEL
LIN {X 0,Y 488.684,Z 254.428,A -85,B 0,C 180,E1 -6516.357,E2 -6516.357} C_VEL
LIN {X 0,Y 488.737,Z 254.415,A -85,B 0,C 180,E1 -6519.251,E2 -6519.251} C_VEL
LIN {X 0,Y 488.707,Z 254.417,A -85,B 0,C 180,E1 -6521.601,E2 -6521.601} C_VEL
LIN {X 0,Y 488.708,Z 254.422,A -85,B 0,C 180,E1 -6524.802,E2 -6524.802} C_VEL
LIN {X 0,Y 488.688,Z 254.42,A -85,B 0,C 180,E1 -6527.475,E2 -6527.475} C_VEL
LIN {X 0,Y 488.73,Z 254.415,A -85,B 0,C 180,E1 -6529.678,E2 -6529.678} C_VEL
LIN {X 0,Y 488.679,Z 254.426,A -85,B 0,C 180,E1 -6532.842,E2 -6532.842} C_VEL
LIN {X 0,Y 488.731,Z 254.417,A -85,B 0,C 180,E1 -6535.888,E2 -6535.888} C_VEL
LIN {X 0,Y 488.691,Z 254.426,A -85,B 0,C 180,E1 -6538.821,E2 -6538.821} C_VEL
LIN {X 0,Y 488.74,Z 254.417,A -85,B 0,C 180,E1 -6541.672,E2 -6541.672} C_VEL
LIN {X 0,Y 488.751,Z 254.414,A -85,B 0,C 180,E1 -6543.529,E2 -6543.529} C_VEL
LIN {X 0,Y 488.758,Z 254.438,A -85,B 0,C 180,E1 -6546.033,E2 -6546.033} C_VEL
LIN {X 0,Y 489.729,Z 260.826,A -85,B 0,C 180,E1 -6547.203,E2 -6547.203} C_VEL
LIN {X 0,Y 489.385,Z 274.61,A -85,B 0,C 180,E1 -6549.62,E2 -6549.62} C_VEL
LIN {X 0,Y 489.026,Z 292.077,A -85,B 0,C 180,E1 -6552.651,E2 -6552.651} C_VEL
LIN {X 0,Y 488.678,Z 310.581,A -85,B 0,C 180,E1 -6555.849,E2 -6555.849} C_VEL
LIN {X 0,Y 488.539,Z 318.6,A -85,B 0,C 180,E1 -6557.207,E2 -6557.207} C_VEL
LIN {X 0,Y 490.193,Z 334.637,A -85,B 0,C 180,E1 -6557.493,E2 -6557.493} C_VEL
LIN {X 0,Y 489.842,Z 396.355,A -85,B 0,C 180,E1 -6558.439,E2 -6558.439} C_VEL
LIN {X 0,Y 489.637,Z 406.155,A -85,B 0,C 180,E1 -6558.696,E2 -6558.696} C_VEL
LIN {X 0,Y 489.37,Z 417.309,A -85,B 0,C 180,E1 -6559.136,E2 -6559.136} C_VEL
LIN {X 0,Y 489.092,Z 428.229,A -85,B 0,C 180,E1 -6559.757,E2 -6559.757} C_VEL
LIN {X 0,Y 488.875,Z 436.705,A -85,B 0,C 180,E1 -6560.38,E2 -6560.38} C_VEL
LIN {X 0,Y 488.628,Z 444.714,A -85,B 0,C 180,E1 -6561.106,E2 -6561.106} C_VEL
LIN {X 0,Y 488.375,Z 452.198,A -85,B 0,C 180,E1 -6561.935,E2 -6561.935} C_VEL
LIN {X 0,Y 488.249,Z 459.804,A -85,B 0,C 180,E1 -6562.973,E2 -6562.973} C_VEL
LIN {X 0,Y 488.088,Z 466.759,A -85,B 0,C 180,E1 -6564.215,E2 -6564.215} C_VEL
LIN {X 0,Y 487.958,Z 472.027,A -85,B 0,C 180,E1 -6565.457,E2 -6565.457} C_VEL
LIN {X 0,Y 488.017,Z 474.735,A -85,B 0,C 180,E1 -6566.285,E2 -6566.285} C_VEL
LIN {X 0,Y 487.962,Z 477.7,A -85,B 0,C 180,E1 -6567.524,E2 -6567.524} C_VEL
LIN {X 0,Y 487.892,Z 478.982,A -85,B 0,C 180,E1 -6568.349,E2 -6568.349} C_VEL
LIN {X 0,Y 487.842,Z 479.782,A -85,B 0,C 180,E1 -6569.175,E2 -6569.175} C_VEL
LIN {X 0,Y 487.836,Z 480.092,A -85,B 0,C 180,E1 -6570,E2 -6570} C_VEL
LIN {X 0,Y 487.841,Z 479.804,A -85,B 0,C 180,E1 -6570.826,E2 -6570.826} C_VEL
LIN {X 0,Y 487.892,Z 479.02,A -85,B 0,C 180,E1 -6571.651,E2 -6571.651} C_VEL
LIN {X 0,Y 487.962,Z 477.754,A -85,B 0,C 180,E1 -6572.477,E2 -6572.477} C_VEL
LIN {X 0,Y 488.017,Z 474.819,A -85,B 0,C 180,E1 -6573.716,E2 -6573.716} C_VEL
LIN {X 0,Y 487.958,Z 472.129,A -85,B 0,C 180,E1 -6574.544,E2 -6574.544} C_VEL
LIN {X 0,Y 488.088,Z 466.887,A -85,B 0,C 180,E1 -6575.785,E2 -6575.785} C_VEL
LIN {X 0,Y 488.242,Z 459.948,A -85,B 0,C 180,E1 -6577.028,E2 -6577.028} C_VEL
LIN {X 0,Y 488.38,Z 452.378,A -85,B 0,C 180,E1 -6578.066,E2 -6578.066} C_VEL
LIN {X 0,Y 488.604,Z 445.943,A -85,B 0,C 180,E1 -6578.791,E2 -6578.791} C_VEL
LIN {X 0,Y 488.862,Z 438.154,A -85,B 0,C 180,E1 -6579.516,E2 -6579.516} C_VEL
LIN {X 0,Y 489.06,Z 429.954,A -85,B 0,C 180,E1 -6580.139,E2 -6580.139} C_VEL
LIN {X 0,Y 489.336,Z 419.555,A -85,B 0,C 180,E1 -6580.761,E2 -6580.761} C_VEL
LIN {X 0,Y 489.578,Z 407.974,A -85,B 0,C 180,E1 -6581.253,E2 -6581.253} C_VEL
LIN {X 0,Y 489.832,Z 397.71,A -85,B 0,C 180,E1 -6581.535,E2 -6581.535} C_VEL
LIN {X 0,Y 490.094,Z 357.808,A -85,B 0,C 180,E1 -6582.156,E2 -6582.156} C_VEL
LIN {X 0,Y 490.042,Z 332.312,A -85,B 0,C 180,E1 -6582.545,E2 -6582.545} C_VEL
LIN {X 0,Y 488.573,Z 319.069,A -85,B 0,C 180,E1 -6582.798,E2 -6582.798} C_VEL
LIN {X 0,Y 488.963,Z 301.837,A -85,B 0,C 180,E1 -6585.848,E2 -6585.848} C_VEL
LIN {X 0,Y 489.397,Z 284.953,A -85,B 0,C 180,E1 -6588.866,E2 -6588.866} C_VEL
LIN {X 0,Y 489.976,Z 267.005,A -85,B 0,C 180,E1 -6592.118,E2 -6592.118} C_VEL
LIN {X 0,Y 490.055,Z 261.925,A -85,B 0,C 180,E1 -6593.053,E2 -6593.053} C_VEL
LIN {X 0,Y 488.73,Z 254.42,A -85,B 0,C 180,E1 -6594.533,E2 -6594.533} C_VEL
LIN {X 0,Y 488.73,Z 254.422,A -85,B 0,C 180,E1 -6597.397,E2 -6597.397} C_VEL
LIN {X 0,Y 488.709,Z 254.417,A -85,B 0,C 180,E1 -6600.362,E2 -6600.362} C_VEL
LIN {X 0,Y 488.734,Z 254.422,A -85,B 0,C 180,E1 -6603.484,E2 -6603.484} C_VEL
LIN {X 0,Y 488.683,Z 254.42,A -85,B 0,C 180,E1 -6606.354,E2 -6606.354} C_VEL
LIN {X 0,Y 488.699,Z 254.423,A -85,B 0,C 180,E1 -6609.254,E2 -6609.254} C_VEL
LIN {X 0,Y 488.707,Z 254.425,A -85,B 0,C 180,E1 -6611.599,E2 -6611.599} C_VEL
LIN {X 0,Y 488.71,Z 254.417,A -85,B 0,C 180,E1 -6614.801,E2 -6614.801} C_VEL
LIN {X 0,Y 488.689,Z 254.427,A -85,B 0,C 180,E1 -6617.474,E2 -6617.474} C_VEL
LIN {X 0,Y 488.731,Z 254.421,A -85,B 0,C 180,E1 -6619.676,E2 -6619.676} C_VEL
LIN {X 0,Y 488.679,Z 254.421,A -85,B 0,C 180,E1 -6622.841,E2 -6622.841} C_VEL
LIN {X 0,Y 488.73,Z 254.418,A -85,B 0,C 180,E1 -6625.887,E2 -6625.887} C_VEL
LIN {X 0,Y 488.688,Z 254.42,A -85,B 0,C 180,E1 -6628.819,E2 -6628.819} C_VEL
LIN {X 0,Y 488.741,Z 254.42,A -85,B 0,C 180,E1 -6631.671,E2 -6631.671} C_VEL
LIN {X 0,Y 488.747,Z 254.412,A -85,B 0,C 180,E1 -6634.444,E2 -6634.444} C_VEL
LIN {X 0,Y 488.724,Z 254.418,A -85,B 0,C 180,E1 -6637.153,E2 -6637.153} C_VEL
LIN {X 0,Y 488.72,Z 254.42,A -85,B 0,C 180,E1 -6639.81,E2 -6639.81} C_VEL
LIN {X 0,Y 488.729,Z 254.415,A -85,B 0,C 180,E1 -6642.423,E2 -6642.423} C_VEL
LIN {X 0,Y 488.756,Z 254.413,A -85,B 0,C 180,E1 -6644.999,E2 -6644.999} C_VEL
LIN {X 0,Y 488.8,Z 254.406,A -85,B 0,C 180,E1 -6648.387,E2 -6648.387} C_VEL
LIN {X 0,Y 488.813,Z 254.41,A -85,B 0,C 180,E1 -6651.733,E2 -6651.733} C_VEL
LIN {X 0,Y 488.849,Z 254.401,A -85,B 0,C 180,E1 -6654.224,E2 -6654.224} C_VEL
LIN {X 0,Y 488.955,Z 254.394,A -85,B 0,C 180,E1 -6657.528,E2 -6657.528} C_VEL
LIN {X 0,Y 488.948,Z 254.388,A -85,B 0,C 180,E1 -6660.823,E2 -6660.823} C_VEL
LIN {X 0,Y 488.955,Z 254.386,A -85,B 0,C 180,E1 -6662.471,E2 -6662.471} C_VEL
LIN {X 0,Y 488.848,Z 254.405,A -85,B 0,C 180,E1 -6665.775,E2 -6665.775} C_VEL
LIN {X 0,Y 488.81,Z 254.405,A -85,B 0,C 180,E1 -6668.266,E2 -6668.266} C_VEL
LIN {X 0,Y 488.822,Z 254.411,A -85,B 0,C 180,E1 -6671.611,E2 -6671.611} C_VEL
LIN {X 0,Y 488.754,Z 254.413,A -85,B 0,C 180,E1 -6675,E2 -6675} C_VEL
LIN {X 0,Y 488.747,Z 254.413,A -85,B 0,C 180,E1 -6678.442,E2 -6678.442} C_VEL
LIN {X 0,Y 488.698,Z 254.421,A -85,B 0,C 180,E1 -6681.07,E2 -6681.07} C_VEL
LIN {X 0,Y 488.684,Z 254.426,A -85,B 0,C 180,E1 -6683.745,E2 -6683.745} C_VEL
LIN {X 0,Y 488.79,Z 254.409,A -85,B 0,C 180,E1 -6686.945,E2 -6686.945} C_VEL
LIN {X 0,Y 488.701,Z 254.419,A -85,B 0,C 180,E1 -6690.362,E2 -6690.362} C_VEL
LIN {X 0,Y 488.727,Z 254.422,A -85,B 0,C 180,E1 -6693.484,E2 -6693.484} C_VEL
LIN {X 0,Y 488.68,Z 254.421,A -85,B 0,C 180,E1 -6696.355,E2 -6696.355} C_VEL
LIN {X 0,Y 488.736,Z 254.418,A -85,B 0,C 180,E1 -6699.25,E2 -6699.25} C_VEL
LIN {X 0,Y 488.685,Z 254.42,A -85,B 0,C 180,E1 -6702.525,E2 -6702.525} C_VEL
LIN {X 0,Y 488.702,Z 254.421,A -85,B 0,C 180,E1 -6705.198,E2 -6705.198} C_VEL
LIN {X 0,Y 488.722,Z 254.422,A -85,B 0,C 180,E1 -6707.478,E2 -6707.478} C_VEL
LIN {X 0,Y 488.733,Z 254.415,A -85,B 0,C 180,E1 -6710.749,E2 -6710.749} C_VEL
LIN {X 0,Y 488.674,Z 254.426,A -85,B 0,C 180,E1 -6713.868,E2 -6713.868} C_VEL
LIN {X 0,Y 488.729,Z 254.416,A -85,B 0,C 180,E1 -6716.877,E2 -6716.877} C_VEL
LIN {X 0,Y 488.714,Z 254.423,A -85,B 0,C 180,E1 -6719.781,E2 -6719.781} C_VEL
LIN {X 0,Y 488.782,Z 254.411,A -85,B 0,C 180,E1 -6723.056,E2 -6723.056} C_VEL
LIN {X 0,Y 488.734,Z 254.414,A -85,B 0,C 180,E1 -6724.356,E2 -6724.356} C_VEL
LIN {X 0,Y 488.092,Z 254.497,A -85,B 0,C 180,E1 -6725.043,E2 -6725.043} C_VEL
LIN {X 0,Y 485.227,Z 254.858,A -85,B 0,C 180,E1 -6726.16,E2 -6726.16} C_VEL
LIN {X 0,Y 482.783,Z 255.164,A -85,B 0,C 180,E1 -6727.06,E2 -6727.06} C_VEL
LIN {X 0,Y 481.726,Z 255.294,A -85,B 0,C 180,E1 -6727.755,E2 -6727.755} C_VEL
LIN {X 0,Y 481.637,Z 255.302,A -85,B 0,C 180,E1 -6727.991,E2 -6727.991} C_VEL
LIN {X 0,Y 481.699,Z 255.291,A -85,B 0,C 180,E1 -6730.393,E2 -6730.393} C_VEL
LIN {X 0,Y 481.682,Z 255.295,A -85,B 0,C 180,E1 -6733.034,E2 -6733.034} C_VEL
LIN {X 0,Y 481.681,Z 255.301,A -85,B 0,C 180,E1 -6735.639,E2 -6735.639} C_VEL
LIN {X 0,Y 481.744,Z 255.287,A -85,B 0,C 180,E1 -6738.215,E2 -6738.215} C_VEL
LIN {X 0,Y 481.754,Z 255.292,A -85,B 0,C 180,E1 -6741.612,E2 -6741.612} C_VEL
LIN {X 0,Y 481.798,Z 255.28,A -85,B 0,C 180,E1 -6744.139,E2 -6744.139} C_VEL
LIN {X 0,Y 481.917,Z 255.27,A -85,B 0,C 180,E1 -6747.492,E2 -6747.492} C_VEL
LIN {X 0,Y 481.896,Z 255.267,A -85,B 0,C 180,E1 -6750.835,E2 -6750.835} C_VEL
LIN {X 0,Y 481.917,Z 255.264,A -85,B 0,C 180,E1 -6752.507,E2 -6752.507} C_VEL
LIN {X 0,Y 481.794,Z 255.284,A -85,B 0,C 180,E1 -6755.86,E2 -6755.86} C_VEL
LIN {X 0,Y 481.751,Z 255.285,A -85,B 0,C 180,E1 -6758.388,E2 -6758.388} C_VEL
LIN {X 0,Y 481.785,Z 255.286,A -85,B 0,C 180,E1 -6761.784,E2 -6761.784} C_VEL
LIN {X 0,Y 481.731,Z 255.29,A -85,B 0,C 180,E1 -6765.224,E2 -6765.224} C_VEL
LIN {X 0,Y 481.701,Z 255.291,A -85,B 0,C 180,E1 -6768.722,E2 -6768.722} C_VEL
LIN {X 0,Y 481.635,Z 255.303,A -85,B 0,C 180,E1 -6771.395,E2 -6771.395} C_VEL
LIN {X 0,Y 481.64,Z 255.301,A -85,B 0,C 180,E1 -6774.114,E2 -6774.114} C_VEL
LIN {X 0,Y 481.703,Z 255.293,A -85,B 0,C 180,E1 -6777.131,E2 -6777.131} C_VEL
LIN {X 0,Y 481.666,Z 255.302,A -85,B 0,C 180,E1 -6779.741,E2 -6779.741} C_VEL
LIN {X 0,Y 481.689,Z 255.402,A -85,B 0,C 180,E1 -6783.014,E2 -6783.014} C_VEL
LIN {X 0,Y 481.553,Z 267.579,A -85,B 0,C 180,E1 -6785.973,E2 -6785.973} C_VEL
LIN {X 0,Y 481.532,Z 268.128,A -85,B 0,C 180,E1 -6786.105,E2 -6786.105} C_VEL
LIN {X 0,Y 483.4,Z 279.123,A -85,B 0,C 180,E1 -6786.33,E2 -6786.33} C_VEL
LIN {X 0,Y 482.958,Z 343.917,A -85,B 0,C 180,E1 -6787.34,E2 -6787.34} C_VEL
LIN {X 0,Y 482.788,Z 353.616,A -85,B 0,C 180,E1 -6787.601,E2 -6787.601} C_VEL
LIN {X 0,Y 482.671,Z 365.086,A -85,B 0,C 180,E1 -6788.07,E2 -6788.07} C_VEL
LIN {X 0,Y 482.393,Z 375.785,A -85,B 0,C 180,E1 -6788.702,E2 -6788.702} C_VEL
LIN {X 0,Y 482.192,Z 383.497,A -85,B 0,C 180,E1 -6789.279,E2 -6789.279} C_VEL
LIN {X 0,Y 481.988,Z 390.447,A -85,B 0,C 180,E1 -6789.908,E2 -6789.908} C_VEL
LIN {X 0,Y 481.726,Z 397.329,A -85,B 0,C 180,E1 -6790.657,E2 -6790.657} C_VEL
LIN {X 0,Y 481.539,Z 403.472,A -85,B 0,C 180,E1 -6791.463,E2 -6791.463} C_VEL
LIN {X 0,Y 481.345,Z 409.436,A -85,B 0,C 180,E1 -6792.415,E2 -6792.415} C_VEL
LIN {X 0,Y 481.192,Z 414.211,A -85,B 0,C 180,E1 -6793.349,E2 -6793.349} C_VEL
LIN {X 0,Y 481.108,Z 418.113,A -85,B 0,C 180,E1 -6794.294,E2 -6794.294} C_VEL
LIN {X 0,Y 480.979,Z 421.825,A -85,B 0,C 180,E1 -6795.465,E2 -6795.465} C_VEL
LIN {X 0,Y 480.873,Z 424.997,A -85,B 0,C 180,E1 -6796.948,E2 -6796.948} C_VEL
LIN {X 0,Y 480.793,Z 426.299,A -85,B 0,C 180,E1 -6798.2,E2 -6798.2} C_VEL
LIN {X 0,Y 480.801,Z 426.484,A -85,B 0,C 180,E1 -6799.471,E2 -6799.471} C_VEL
LIN {X 0,Y 480.811,Z 425.51,A -85,B 0,C 180,E1 -6800.776,E2 -6800.776} C_VEL
LIN {X 0,Y 480.929,Z 423.22,A -85,B 0,C 180,E1 -6802.139,E2 -6802.139} C_VEL
LIN {X 0,Y 481.066,Z 419.499,A -85,B 0,C 180,E1 -6803.464,E2 -6803.464} C_VEL
LIN {X 0,Y 481.206,Z 415.135,A -85,B 0,C 180,E1 -6804.588,E2 -6804.588} C_VEL
LIN {X 0,Y 481.376,Z 410.419,A -85,B 0,C 180,E1 -6805.548,E2 -6805.548} C_VEL
LIN {X 0,Y 481.5,Z 405.889,A -85,B 0,C 180,E1 -6806.315,E2 -6806.315} C_VEL
LIN {X 0,Y 481.694,Z 399.526,A -85,B 0,C 180,E1 -6807.204,E2 -6807.204} C_VEL
LIN {X 0,Y 481.958,Z 393.239,A -85,B 0,C 180,E1 -6807.934,E2 -6807.934} C_VEL
LIN {X 0,Y 482.163,Z 386.454,A -85,B 0,C 180,E1 -6808.595,E2 -6808.595} C_VEL
LIN {X 0,Y 482.434,Z 378.12,A -85,B 0,C 180,E1 -6809.258,E2 -6809.258} C_VEL
LIN {X 0,Y 482.563,Z 370.032,A -85,B 0,C 180,E1 -6809.778,E2 -6809.778} C_VEL
LIN {X 0,Y 482.735,Z 361.446,A -85,B 0,C 180,E1 -6810.212,E2 -6810.212} C_VEL
LIN {X 0,Y 482.899,Z 351.775,A -85,B 0,C 180,E1 -6810.572,E2 -6810.572} C_VEL
LIN {X 0,Y 482.978,Z 341.844,A -85,B 0,C 180,E1 -6810.816,E2 -6810.816} C_VEL
LIN {X 0,Y 483.433,Z 278.045,A -85,B 0,C 180,E1 -6811.806,E2 -6811.806} C_VEL
LIN {X 0,Y 481.63,Z 267.977,A -85,B 0,C 180,E1 -6812.017,E2 -6812.017} C_VEL
LIN {X 0,Y 481.574,Z 255.314,A -85,B 0,C 180,E1 -6814.615,E2 -6814.615} C_VEL
LIN {X 0,Y 481.636,Z 255.303,A -85,B 0,C 180,E1 -6817.705,E2 -6817.705} C_VEL
LIN {X 0,Y 481.697,Z 255.302,A -85,B 0,C 180,E1 -6820.394,E2 -6820.394} C_VEL
LIN {X 0,Y 481.681,Z 255.296,A -85,B 0,C 180,E1 -6823.034,E2 -6823.034} C_VEL
LIN {X 0,Y 481.678,Z 255.294,A -85,B 0,C 180,E1 -6825.639,E2 -6825.639} C_VEL
LIN {X 0,Y 481.742,Z 255.291,A -85,B 0,C 180,E1 -6828.216,E2 -6828.216} C_VEL
LIN {X 0,Y 481.753,Z 255.285,A -85,B 0,C 180,E1 -6831.612,E2 -6831.612} C_VEL
LIN {X 0,Y 481.812,Z 255.281,A -85,B 0,C 180,E1 -6834.14,E2 -6834.14} C_VEL
LIN {X 0,Y 481.919,Z 255.262,A -85,B 0,C 180,E1 -6837.493,E2 -6837.493} C_VEL
LIN {X 0,Y 481.916,Z 255.266,A -85,B 0,C 180,E1 -6840.836,E2 -6840.836} C_VEL
LIN {X 0,Y 481.92,Z 255.271,A -85,B 0,C 180,E1 -6842.508,E2 -6842.508} C_VEL
LIN {X 0,Y 481.808,Z 255.278,A -85,B 0,C 180,E1 -6845.861,E2 -6845.861} C_VEL
LIN {X 0,Y 481.755,Z 255.287,A -85,B 0,C 180,E1 -6848.389,E2 -6848.389} C_VEL
LIN {X 0,Y 481.742,Z 255.285,A -85,B 0,C 180,E1 -6851.786,E2 -6851.786} C_VEL
LIN {X 0,Y 481.736,Z 255.286,A -85,B 0,C 180,E1 -6855.225,E2 -6855.225} C_VEL
LIN {X 0,Y 481.705,Z 255.294,A -85,B 0,C 180,E1 -6858.723,E2 -6858.723} C_VEL
LIN {X 0,Y 481.64,Z 255.295,A -85,B 0,C 180,E1 -6861.396,E2 -6861.396} C_VEL
LIN {X 0,Y 481.67,Z 255.297,A -85,B 0,C 180,E1 -6864.114,E2 -6864.114} C_VEL
LIN {X 0,Y 481.746,Z 255.286,A -85,B 0,C 180,E1 -6867.141,E2 -6867.141} C_VEL
LIN {X 0,Y 481.682,Z 255.289,A -85,B 0,C 180,E1 -6869.741,E2 -6869.741} C_VEL
LIN {X 0,Y 481.666,Z 255.297,A -85,B 0,C 180,E1 -6872.675,E2 -6872.675} C_VEL
LIN {X 0,Y 481.638,Z 255.299,A -85,B 0,C 180,E1 -6875.71,E2 -6875.71} C_VEL
LIN {X 0,Y 481.709,Z 255.29,A -85,B 0,C 180,E1 -6879.355,E2 -6879.355} C_VEL
LIN {X 0,Y 481.644,Z 255.301,A -85,B 0,C 180,E1 -6882.162,E2 -6882.162} C_VEL
LIN {X 0,Y 481.656,Z 255.297,A -85,B 0,C 180,E1 -6885.544,E2 -6885.544} C_VEL
LIN {X 0,Y 481.653,Z 255.299,A -85,B 0,C 180,E1 -6888.959,E2 -6888.959} C_VEL
LIN {X 0,Y 481.652,Z 255.299,A -85,B 0,C 180,E1 -6891.994,E2 -6891.994} C_VEL
LIN {X 0,Y 481.69,Z 255.293,A -85,B 0,C 180,E1 -6895.319,E2 -6895.319} C_VEL
LIN {X 0,Y 481.644,Z 255.304,A -85,B 0,C 180,E1 -6898.312,E2 -6898.312} C_VEL
LIN {X 0,Y 481.696,Z 255.295,A -85,B 0,C 180,E1 -6901.219,E2 -6901.219} C_VEL
LIN {X 0,Y 481.688,Z 255.297,A -85,B 0,C 180,E1 -6904.043,E2 -6904.043} C_VEL
LIN {X 0,Y 481.732,Z 255.379,A -85,B 0,C 180,E1 -6905.918,E2 -6905.918} C_VEL
LIN {X 0,Y 482.698,Z 261.611,A -85,B 0,C 180,E1 -6907.079,E2 -6907.079} C_VEL
LIN {X 0,Y 482.448,Z 274.267,A -85,B 0,C 180,E1 -6909.332,E2 -6909.332} C_VEL
LIN {X 0,Y 481.975,Z 292.878,A -85,B 0,C 180,E1 -6912.608,E2 -6912.608} C_VEL
LIN {X 0,Y 481.603,Z 311.417,A -85,B 0,C 180,E1 -6915.852,E2 -6915.852} C_VEL
LIN {X 0,Y 481.494,Z 318.168,A -85,B 0,C 180,E1 -6917.01,E2 -6917.01} C_VEL
LIN {X 0,Y 483.263,Z 336.109,A -85,B 0,C 180,E1 -6917.339,E2 -6917.339} C_VEL
LIN {X 0,Y 482.887,Z 395.827,A -85,B 0,C 180,E1 -6918.27,E2 -6918.27} C_VEL
LIN {X 0,Y 482.649,Z 405.661,A -85,B 0,C 180,E1 -6918.531,E2 -6918.531} C_VEL
LIN {X 0,Y 482.342,Z 416.837,A -85,B 0,C 180,E1 -6918.975,E2 -6918.975} C_VEL
LIN {X 0,Y 482.087,Z 427.78,A -85,B 0,C 180,E1 -6919.607,E2 -6919.607} C_VEL
LIN {X 0,Y 481.815,Z 436.262,A -85,B 0,C 180,E1 -6920.238,E2 -6920.238} C_VEL
LIN {X 0,Y 481.581,Z 444.282,A -85,B 0,C 180,E1 -6920.974,E2 -6920.974} C_VEL
LIN {X 0,Y 481.316,Z 451.775,A -85,B 0,C 180,E1 -6921.816,E2 -6921.816} C_VEL
LIN {X 0,Y 481.173,Z 459.388,A -85,B 0,C 180,E1 -6922.869,E2 -6922.869} C_VEL
LIN {X 0,Y 480.992,Z 466.35,A -85,B 0,C 180,E1 -6924.13,E2 -6924.13} C_VEL
LIN {X 0,Y 480.874,Z 471.626,A -85,B 0,C 180,E1 -6925.39,E2 -6925.39} C_VEL
LIN {X 0,Y 480.939,Z 474.336,A -85,B 0,C 180,E1 -6926.23,E2 -6926.23} C_VEL
LIN {X 0,Y 480.872,Z 477.305,A -85,B 0,C 180,E1 -6927.487,E2 -6927.487} C_VEL
LIN {X 0,Y 480.824,Z 478.589,A -85,B 0,C 180,E1 -6928.325,E2 -6928.325} C_VEL
LIN {X 0,Y 480.767,Z 479.39,A -85,B 0,C 180,E1 -6929.163,E2 -6929.163} C_VEL
LIN {X 0,Y 480.759,Z 479.701,A -85,B 0,C 180,E1 -6930,E2 -6930} C_VEL
LIN {X 0,Y 480.767,Z 479.413,A -85,B 0,C 180,E1 -6930.838,E2 -6930.838} C_VEL
LIN {X 0,Y 480.824,Z 478.626,A -85,B 0,C 180,E1 -6931.675,E2 -6931.675} C_VEL
LIN {X 0,Y 480.872,Z 477.357,A -85,B 0,C 180,E1 -6932.513,E2 -6932.513} C_VEL
LIN {X 0,Y 480.939,Z 474.418,A -85,B 0,C 180,E1 -6933.771,E2 -6933.771} C_VEL
LIN {X 0,Y 480.874,Z 471.721,A -85,B 0,C 180,E1 -6934.611,E2 -6934.611} C_VEL
LIN {X 0,Y 480.992,Z 466.471,A -85,B 0,C 180,E1 -6935.871,E2 -6935.871} C_VEL
LIN {X 0,Y 481.169,Z 459.515,A -85,B 0,C 180,E1 -6937.132,E2 -6937.132} C_VEL
LIN {X 0,Y 481.322,Z 451.934,A -85,B 0,C 180,E1 -6938.185,E2 -6938.185} C_VEL
LIN {X 0,Y 481.55,Z 445.485,A -85,B 0,C 180,E1 -6938.921,E2 -6938.921} C_VEL
LIN {X 0,Y 481.835,Z 437.68,A -85,B 0,C 180,E1 -6939.656,E2 -6939.656} C_VEL
LIN {X 0,Y 482.043,Z 429.459,A -85,B 0,C 180,E1 -6940.288,E2 -6940.288} C_VEL
LIN {X 0,Y 482.257,Z 420.907,A -85,B 0,C 180,E1 -6940.814,E2 -6940.814} C_VEL
LIN {X 0,Y 482.56,Z 409.666,A -85,B 0,C 180,E1 -6941.339,E2 -6941.339} C_VEL
LIN {X 0,Y 482.836,Z 398.236,A -85,B 0,C 180,E1 -6941.678,E2 -6941.678} C_VEL
LIN {X 0,Y 483.055,Z 374.391,A -85,B 0,C 180,E1 -6942.069,E2 -6942.069} C_VEL
LIN {X 0,Y 483.079,Z 332.721,A -85,B 0,C 180,E1 -6942.711,E2 -6942.711} C_VEL
LIN {X 0,Y 481.539,Z 318.703,A -85,B 0,C 180,E1 -6942.986,E2 -6942.986} C_VEL
LIN {X 0,Y 481.915,Z 302.47,A -85,B 0,C 180,E1 -6945.903,E2 -6945.903} C_VEL
LIN {X 0,Y 482.383,Z 285.991,A -85,B 0,C 180,E1 -6948.893,E2 -6948.893} C_VEL
LIN {X 0,Y 483.001,Z 267.845,A -85,B 0,C 180,E1 -6952.229,E2 -6952.229} C_VEL
LIN {X 0,Y 483.068,Z 263.024,A -85,B 0,C 180,E1 -6953.129,E2 -6953.129} C_VEL
LIN {X 0,Y 481.703,Z 255.296,A -85,B 0,C 180,E1 -6954.685,E2 -6954.685} C_VEL
LIN {X 0,Y 481.692,Z 255.297,A -85,B 0,C 180,E1 -6957.832,E2 -6957.832} C_VEL
LIN {X 0,Y 481.645,Z 255.297,A -85,B 0,C 180,E1 -6960.711,E2 -6960.711} C_VEL
LIN {X 0,Y 481.697,Z 255.296,A -85,B 0,C 180,E1 -6963.733,E2 -6963.733} C_VEL
LIN {X 0,Y 481.625,Z 255.3,A -85,B 0,C 180,E1 -6966.746,E2 -6966.746} C_VEL
LIN {X 0,Y 481.676,Z 255.296,A -85,B 0,C 180,E1 -6969.94,E2 -6969.94} C_VEL
LIN {X 0,Y 481.638,Z 255.303,A -85,B 0,C 180,E1 -6973.299,E2 -6973.299} C_VEL
LIN {X 0,Y 481.656,Z 255.303,A -85,B 0,C 180,E1 -6975.64,E2 -6975.64} C_VEL
LIN {X 0,Y 481.655,Z 255.297,A -85,B 0,C 180,E1 -6978.958,E2 -6978.958} C_VEL
LIN {X 0,Y 481.653,Z 255.298,A -85,B 0,C 180,E1 -6981.992,E2 -6981.992} C_VEL
LIN {X 0,Y 481.689,Z 255.297,A -85,B 0,C 180,E1 -6985.317,E2 -6985.317} C_VEL
LIN {X 0,Y 481.641,Z 255.298,A -85,B 0,C 180,E1 -6988.311,E2 -6988.311} C_VEL
LIN {X 0,Y 481.696,Z 255.294,A -85,B 0,C 180,E1 -6991.218,E2 -6991.218} C_VEL
LIN {X 0,Y 481.703,Z 255.292,A -85,B 0,C 180,E1 -6994.042,E2 -6994.042} C_VEL
LIN {X 0,Y 481.67,Z 255.294,A -85,B 0,C 180,E1 -6996.811,E2 -6996.811} C_VEL
LIN {X 0,Y 481.691,Z 255.299,A -85,B 0,C 180,E1 -6999.502,E2 -6999.502} C_VEL
LIN {X 0,Y 481.702,Z 255.291,A -85,B 0,C 180,E1 -7002.158,E2 -7002.158} C_VEL
LIN {X 0,Y 481.737,Z 255.286,A -85,B 0,C 180,E1 -7004.775,E2 -7004.775} C_VEL
LIN {X 0,Y 481.745,Z 255.286,A -85,B 0,C 180,E1 -7008.214,E2 -7008.214} C_VEL
LIN {X 0,Y 481.758,Z 255.291,A -85,B 0,C 180,E1 -7011.611,E2 -7011.611} C_VEL
LIN {X 0,Y 481.81,Z 255.278,A -85,B 0,C 180,E1 -7014.139,E2 -7014.139} C_VEL
LIN {X 0,Y 481.922,Z 255.27,A -85,B 0,C 180,E1 -7017.492,E2 -7017.492} C_VEL
LIN {X 0,Y 481.899,Z 255.266,A -85,B 0,C 180,E1 -7020.835,E2 -7020.835} C_VEL
LIN {X 0,Y 481.922,Z 255.263,A -85,B 0,C 180,E1 -7022.507,E2 -7022.507} C_VEL
LIN {X 0,Y 481.809,Z 255.281,A -85,B 0,C 180,E1 -7025.86,E2 -7025.86} C_VEL
LIN {X 0,Y 481.756,Z 255.284,A -85,B 0,C 180,E1 -7028.388,E2 -7028.388} C_VEL
LIN {X 0,Y 481.787,Z 255.285,A -85,B 0,C 180,E1 -7031.783,E2 -7031.783} C_VEL
LIN {X 0,Y 481.734,Z 255.29,A -85,B 0,C 180,E1 -7035.224,E2 -7035.224} C_VEL
LIN {X 0,Y 481.704,Z 255.29,A -85,B 0,C 180,E1 -7038.721,E2 -7038.721} C_VEL
LIN {X 0,Y 481.637,Z 255.304,A -85,B 0,C 180,E1 -7041.394,E2 -7041.394} C_VEL
LIN {X 0,Y 481.668,Z 255.296,A -85,B 0,C 180,E1 -7044.113,E2 -7044.113} C_VEL
LIN {X 0,Y 481.743,Z 255.288,A -85,B 0,C 180,E1 -7047.14,E2 -7047.14} C_VEL
LIN {X 0,Y 481.67,Z 255.3,A -85,B 0,C 180,E1 -7049.741,E2 -7049.741} C_VEL
LIN {X 0,Y 481.664,Z 255.295,A -85,B 0,C 180,E1 -7052.674,E2 -7052.674} C_VEL
LIN {X 0,Y 481.634,Z 255.305,A -85,B 0,C 180,E1 -7055.708,E2 -7055.708} C_VEL
LIN {X 0,Y 481.707,Z 255.294,A -85,B 0,C 180,E1 -7059.354,E2 -7059.354} C_VEL
LIN {X 0,Y 481.645,Z 255.299,A -85,B 0,C 180,E1 -7062.16,E2 -7062.16} C_VEL
LIN {X 0,Y 481.651,Z 255.304,A -85,B 0,C 180,E1 -7065.542,E2 -7065.542} C_VEL
LIN {X 0,Y 481.664,Z 255.297,A -85,B 0,C 180,E1 -7068.084,E2 -7068.084} C_VEL
LIN {X 0,Y 481.688,Z 255.295,A -85,B 0,C 180,E1 -7071.143,E2 -7071.143} C_VEL
LIN {X 0,Y 481.657,Z 255.296,A -85,B 0,C 180,E1 -7074.795,E2 -7074.795} C_VEL
LIN {X 0,Y 481.663,Z 255.299,A -85,B 0,C 180,E1 -7077.326,E2 -7077.326} C_VEL
LIN {X 0,Y 481.669,Z 255.295,A -85,B 0,C 180,E1 -7080.259,E2 -7080.259} C_VEL
LIN {X 0,Y 481.736,Z 255.289,A -85,B 0,C 180,E1 -7083.112,E2 -7083.112} C_VEL
LIN {X 0,Y 481.673,Z 255.298,A -85,B 0,C 180,E1 -7085.887,E2 -7085.887} C_VEL
LIN {X 0,Y 481.637,Z 255.302,A -85,B 0,C 180,E1 -7087.991,E2 -7087.991} C_VEL
LIN {X 0,Y 480.967,Z 255.382,A -85,B 0,C 180,E1 -7088.689,E2 -7088.689} C_VEL
LIN {X 0,Y 478.136,Z 255.74,A -85,B 0,C 180,E1 -7089.823,E2 -7089.823} C_VEL
LIN {X 0,Y 475.749,Z 256.037,A -85,B 0,C 180,E1 -7090.737,E2 -7090.737} C_VEL
LIN {X 0,Y 474.728,Z 256.165,A -85,B 0,C 180,E1 -7091.443,E2 -7091.443} C_VEL
LIN {X 0,Y 474.646,Z 256.173,A -85,B 0,C 180,E1 -7091.682,E2 -7091.682} C_VEL
LIN {X 0,Y 474.691,Z 256.164,A -85,B 0,C 180,E1 -7094.544,E2 -7094.544} C_VEL
LIN {X 0,Y 474.696,Z 256.166,A -85,B 0,C 180,E1 -7098.037,E2 -7098.037} C_VEL
LIN {X 0,Y 474.719,Z 256.166,A -85,B 0,C 180,E1 -7101.486,E2 -7101.486} C_VEL
LIN {X 0,Y 474.76,Z 256.158,A -85,B 0,C 180,E1 -7104.052,E2 -7104.052} C_VEL
LIN {X 0,Y 474.883,Z 256.145,A -85,B 0,C 180,E1 -7107.455,E2 -7107.455} C_VEL
LIN {X 0,Y 474.848,Z 256.145,A -85,B 0,C 180,E1 -7110.848,E2 -7110.848} C_VEL
LIN {X 0,Y 474.883,Z 256.14,A -85,B 0,C 180,E1 -7112.544,E2 -7112.544} C_VEL
LIN {X 0,Y 474.757,Z 256.16,A -85,B 0,C 180,E1 -7115.948,E2 -7115.948} C_VEL
LIN {X 0,Y 474.717,Z 256.161,A -85,B 0,C 180,E1 -7118.513,E2 -7118.513} C_VEL
LIN {X 0,Y 474.729,Z 256.163,A -85,B 0,C 180,E1 -7121.961,E2 -7121.961} C_VEL
LIN {X 0,Y 474.67,Z 256.173,A -85,B 0,C 180,E1 -7125.767,E2 -7125.767} C_VEL
LIN {X 0,Y 474.653,Z 256.171,A -85,B 0,C 180,E1 -7129.01,E2 -7129.01} C_VEL
LIN {X 0,Y 474.577,Z 256.185,A -85,B 0,C 180,E1 -7131.729,E2 -7131.729} C_VEL
LIN {X 0,Y 474.618,Z 256.173,A -85,B 0,C 180,E1 -7134.494,E2 -7134.494} C_VEL
LIN {X 0,Y 474.662,Z 256.171,A -85,B 0,C 180,E1 -7137.332,E2 -7137.332} C_VEL
LIN {X 0,Y 474.592,Z 256.178,A -85,B 0,C 180,E1 -7140.23,E2 -7140.23} C_VEL
LIN {X 0,Y 474.636,Z 256.29,A -85,B 0,C 180,E1 -7142.947,E2 -7142.947} C_VEL
LIN {X 0,Y 474.529,Z 266.545,A -85,B 0,C 180,E1 -7145.457,E2 -7145.457} C_VEL
LIN {X 0,Y 474.545,Z 268.406,A -85,B 0,C 180,E1 -7145.91,E2 -7145.91} C_VEL
LIN {X 0,Y 476.472,Z 280.033,A -85,B 0,C 180,E1 -7146.156,E2 -7146.156} C_VEL
LIN {X 0,Y 476.015,Z 344.309,A -85,B 0,C 180,E1 -7147.175,E2 -7147.175} C_VEL
LIN {X 0,Y 475.854,Z 354.243,A -85,B 0,C 180,E1 -7147.449,E2 -7147.449} C_VEL
LIN {X 0,Y 475.691,Z 366.096,A -85,B 0,C 180,E1 -7147.949,E2 -7147.949} C_VEL
LIN {X 0,Y 475.411,Z 375.388,A -85,B 0,C 180,E1 -7148.501,E2 -7148.501} C_VEL
LIN {X 0,Y 475.221,Z 383.114,A -85,B 0,C 180,E1 -7149.076,E2 -7149.076} C_VEL
LIN {X 0,Y 475.02,Z 390.115,A -85,B 0,C 180,E1 -7149.706,E2 -7149.706} C_VEL
LIN {X 0,Y 474.712,Z 397.584,A -85,B 0,C 180,E1 -7150.525,E2 -7150.525} C_VEL
LIN {X 0,Y 474.524,Z 403.775,A -85,B 0,C 180,E1 -7151.346,E2 -7151.346} C_VEL
LIN {X 0,Y 474.334,Z 409.139,A -85,B 0,C 180,E1 -7152.2,E2 -7152.2} C_VEL
LIN {X 0,Y 474.193,Z 413.29,A -85,B 0,C 180,E1 -7152.98,E2 -7152.98} C_VEL
LIN {X 0,Y 474.058,Z 418.282,A -85,B 0,C 180,E1 -7154.168,E2 -7154.168} C_VEL
LIN {X 0,Y 473.909,Z 422.12,A -85,B 0,C 180,E1 -7155.383,E2 -7155.383} C_VEL
LIN {X 0,Y 473.805,Z 424.849,A -85,B 0,C 180,E1 -7156.619,E2 -7156.619} C_VEL
LIN {X 0,Y 473.725,Z 426.661,A -85,B 0,C 180,E1 -7158.119,E2 -7158.119} C_VEL
LIN {X 0,Y 473.729,Z 426.958,A -85,B 0,C 180,E1 -7159.251,E2 -7159.251} C_VEL
LIN {X 0,Y 473.712,Z 426.259,A -85,B 0,C 180,E1 -7160.485,E2 -7160.485} C_VEL
LIN {X 0,Y 473.823,Z 424.303,A -85,B 0,C 180,E1 -7161.823,E2 -7161.823} C_VEL
LIN {X 0,Y 473.977,Z 420.985,A -85,B 0,C 180,E1 -7163.195,E2 -7163.195} C_VEL
LIN {X 0,Y 474.093,Z 417.696,A -85,B 0,C 180,E1 -7164.153,E2 -7164.153} C_VEL
LIN {X 0,Y 474.314,Z 411.741,A -85,B 0,C 180,E1 -7165.477,E2 -7165.477} C_VEL
LIN {X 0,Y 474.479,Z 406.357,A -85,B 0,C 180,E1 -7166.414,E2 -7166.414} C_VEL
LIN {X 0,Y 474.647,Z 400.992,A -85,B 0,C 180,E1 -7167.194,E2 -7167.194} C_VEL
LIN {X 0,Y 474.977,Z 393.67,A -85,B 0,C 180,E1 -7168.065,E2 -7168.065} C_VEL
LIN {X 0,Y 475.224,Z 385.826,A -85,B 0,C 180,E1 -7168.829,E2 -7168.829} C_VEL
LIN {X 0,Y 475.508,Z 377.766,A -85,B 0,C 180,E1 -7169.466,E2 -7169.466} C_VEL
LIN {X 0,Y 475.616,Z 370.329,A -85,B 0,C 180,E1 -7169.947,E2 -7169.947} C_VEL
LIN {X 0,Y 475.793,Z 361.921,A -85,B 0,C 180,E1 -7170.377,E2 -7170.377} C_VEL
LIN {X 0,Y 475.962,Z 352.428,A -85,B 0,C 180,E1 -7170.738,E2 -7170.738} C_VEL
LIN {X 0,Y 476.047,Z 342.138,A -85,B 0,C 180,E1 -7170.997,E2 -7170.997} C_VEL
LIN {X 0,Y 476.524,Z 278.666,A -85,B 0,C 180,E1 -7171.997,E2 -7171.997} C_VEL
LIN {X 0,Y 474.642,Z 268.206,A -85,B 0,C 180,E1 -7172.231,E2 -7172.231} C_VEL
LIN {X 0,Y 474.566,Z 256.187,A -85,B 0,C 180,E1 -7174.76,E2 -7174.76} C_VEL
LIN {X 0,Y 474.58,Z 256.182,A -85,B 0,C 180,E1 -7177.355,E2 -7177.355} C_VEL
LIN {X 0,Y 474.645,Z 256.177,A -85,B 0,C 180,E1 -7180.09,E2 -7180.09} C_VEL
LIN {X 0,Y 474.64,Z 256.176,A -85,B 0,C 180,E1 -7182.775,E2 -7182.775} C_VEL
LIN {X 0,Y 474.637,Z 256.172,A -85,B 0,C 180,E1 -7185.422,E2 -7185.422} C_VEL
LIN {X 0,Y 474.694,Z 256.167,A -85,B 0,C 180,E1 -7188.038,E2 -7188.038} C_VEL
LIN {X 0,Y 474.719,Z 256.162,A -85,B 0,C 180,E1 -7191.487,E2 -7191.487} C_VEL
LIN {X 0,Y 474.773,Z 256.157,A -85,B 0,C 180,E1 -7194.053,E2 -7194.053} C_VEL
LIN {X 0,Y 474.886,Z 256.138,A -85,B 0,C 180,E1 -7197.456,E2 -7197.456} C_VEL
LIN {X 0,Y 474.867,Z 256.144,A -85,B 0,C 180,E1 -7200.849,E2 -7200.849} C_VEL
LIN {X 0,Y 474.886,Z 256.147,A -85,B 0,C 180,E1 -7202.545,E2 -7202.545} C_VEL
LIN {X 0,Y 474.77,Z 256.155,A -85,B 0,C 180,E1 -7205.948,E2 -7205.948} C_VEL
LIN {X 0,Y 474.72,Z 256.164,A -85,B 0,C 180,E1 -7208.514,E2 -7208.514} C_VEL
LIN {X 0,Y 474.695,Z 256.164,A -85,B 0,C 180,E1 -7211.963,E2 -7211.963} C_VEL
LIN {X 0,Y 474.692,Z 256.163,A -85,B 0,C 180,E1 -7215.456,E2 -7215.456} C_VEL
LIN {X 0,Y 474.658,Z 256.169,A -85,B 0,C 180,E1 -7219.011,E2 -7219.011} C_VEL
LIN {X 0,Y 474.582,Z 256.174,A -85,B 0,C 180,E1 -7221.73,E2 -7221.73} C_VEL
LIN {X 0,Y 474.652,Z 256.172,A -85,B 0,C 180,E1 -7224.494,E2 -7224.494} C_VEL
LIN {X 0,Y 474.693,Z 256.164,A -85,B 0,C 180,E1 -7227.34,E2 -7227.34} C_VEL
LIN {X 0,Y 474.603,Z 256.179,A -85,B 0,C 180,E1 -7230.812,E2 -7230.812} C_VEL
LIN {X 0,Y 474.633,Z 256.169,A -85,B 0,C 180,E1 -7233.985,E2 -7233.985} C_VEL
LIN {X 0,Y 474.57,Z 256.179,A -85,B 0,C 180,E1 -7236.901,E2 -7236.901} C_VEL
LIN {X 0,Y 474.646,Z 256.17,A -85,B 0,C 180,E1 -7239.652,E2 -7239.652} C_VEL
LIN {X 0,Y 474.602,Z 256.176,A -85,B 0,C 180,E1 -7242.936,E2 -7242.936} C_VEL
LIN {X 0,Y 474.605,Z 256.176,A -85,B 0,C 180,E1 -7245.896,E2 -7245.896} C_VEL
LIN {X 0,Y 474.624,Z 256.174,A -85,B 0,C 180,E1 -7249.042,E2 -7249.042} C_VEL
LIN {X 0,Y 474.607,Z 256.175,A -85,B 0,C 180,E1 -7251.705,E2 -7251.705} C_VEL
LIN {X 0,Y 474.626,Z 256.178,A -85,B 0,C 180,E1 -7254.727,E2 -7254.727} C_VEL
LIN {X 0,Y 474.634,Z 256.173,A -85,B 0,C 180,E1 -7257.789,E2 -7257.789} C_VEL
LIN {X 0,Y 474.621,Z 256.179,A -85,B 0,C 180,E1 -7260.886,E2 -7260.886} C_VEL
LIN {X 0,Y 474.652,Z 256.171,A -85,B 0,C 180,E1 -7263.629,E2 -7263.629} C_VEL
LIN {X 0,Y 474.696,Z 256.334,A -85,B 0,C 180,E1 -7265.801,E2 -7265.801} C_VEL
LIN {X 0,Y 475.741,Z 263.661,A -85,B 0,C 180,E1 -7267.184,E2 -7267.184} C_VEL
LIN {X 0,Y 475.325,Z 278.712,A -85,B 0,C 180,E1 -7269.894,E2 -7269.894} C_VEL
LIN {X 0,Y 474.855,Z 298.638,A -85,B 0,C 180,E1 -7273.447,E2 -7273.447} C_VEL
LIN {X 0,Y 474.489,Z 316.059,A -85,B 0,C 180,E1 -7276.532,E2 -7276.532} C_VEL
LIN {X 0,Y 474.458,Z 317.551,A -85,B 0,C 180,E1 -7276.795,E2 -7276.795} C_VEL
LIN {X 0,Y 476.343,Z 335.431,A -85,B 0,C 180,E1 -7277.141,E2 -7277.141} C_VEL
LIN {X 0,Y 475.945,Z 395.483,A -85,B 0,C 180,E1 -7278.097,E2 -7278.097} C_VEL
LIN {X 0,Y 475.699,Z 405.271,A -85,B 0,C 180,E1 -7278.361,E2 -7278.361} C_VEL
LIN {X 0,Y 475.372,Z 416.421,A -85,B 0,C 180,E1 -7278.812,E2 -7278.812} C_VEL
LIN {X 0,Y 475.083,Z 427.353,A -85,B 0,C 180,E1 -7279.452,E2 -7279.452} C_VEL
LIN {X 0,Y 474.788,Z 435.83,A -85,B 0,C 180,E1 -7280.092,E2 -7280.092} C_VEL
LIN {X 0,Y 474.508,Z 443.85,A -85,B 0,C 180,E1 -7280.839,E2 -7280.839} C_VEL
LIN {X 0,Y 474.274,Z 451.354,A -85,B 0,C 180,E1 -7281.693,E2 -7281.693} C_VEL
LIN {X 0,Y 474.11,Z 458.973,A -85,B 0,C 180,E1 -7282.762,E2 -7282.762} C_VEL
LIN {X 0,Y 473.9,Z 465.941,A -85,B 0,C 180,E1 -7284.042,E2 -7284.042} C_VEL
LIN {X 0,Y 473.796,Z 471.226,A -85,B 0,C 180,E1 -7285.321,E2 -7285.321} C_VEL
LIN {X 0,Y 473.849,Z 475.121,A -85,B 0,C 180,E1 -7286.599,E2 -7286.599} C_VEL
LIN {X 0,Y 473.787,Z 476.912,A -85,B 0,C 180,E1 -7287.45,E2 -7287.45} C_VEL
LIN {X 0,Y 473.757,Z 478.198,A -85,B 0,C 180,E1 -7288.3,E2 -7288.3} C_VEL
LIN {X 0,Y 473.695,Z 478.999,A -85,B 0,C 180,E1 -7289.15,E2 -7289.15} C_VEL
LIN {X 0,Y 473.684,Z 479.31,A -85,B 0,C 180,E1 -7290,E2 -7290} C_VEL
LIN {X 0,Y 473.695,Z 479.022,A -85,B 0,C 180,E1 -7290.85,E2 -7290.85} C_VEL
LIN {X 0,Y 473.757,Z 478.234,A -85,B 0,C 180,E1 -7291.7,E2 -7291.7} C_VEL
LIN {X 0,Y 473.787,Z 476.959,A -85,B 0,C 180,E1 -7292.551,E2 -7292.551} C_VEL
LIN {X 0,Y 473.843,Z 474.015,A -85,B 0,C 180,E1 -7293.827,E2 -7293.827} C_VEL
LIN {X 0,Y 473.796,Z 471.314,A -85,B 0,C 180,E1 -7294.68,E2 -7294.68} C_VEL
LIN {X 0,Y 473.901,Z 467.991,A -85,B 0,C 180,E1 -7295.532,E2 -7295.532} C_VEL
LIN {X 0,Y 474.026,Z 462.714,A -85,B 0,C 180,E1 -7296.608,E2 -7296.608} C_VEL
LIN {X 0,Y 474.135,Z 456.22,A -85,B 0,C 180,E1 -7297.666,E2 -7297.666} C_VEL
LIN {X 0,Y 474.416,Z 448.043,A -85,B 0,C 180,E1 -7298.734,E2 -7298.734} C_VEL
LIN {X 0,Y 474.771,Z 438.444,A -85,B 0,C 180,E1 -7299.694,E2 -7299.694} C_VEL
LIN {X 0,Y 474.992,Z 430.472,A -85,B 0,C 180,E1 -7300.335,E2 -7300.335} C_VEL
